LIN {X 0,Y 560.232,Z 513.242,A -85,B 0,C 180,E1 26436.285,E2 26436.285} C_VEL
LIN {X 0,Y 559.276,Z 513.366,A -85,B 0,C 180,E1 26435.497,E2 26435.497} C_VEL
LIN {X 0,Y 552.777,Z 514.194,A -85,B 0,C 180,E1 26433.228,E2 26433.228} C_VEL
LIN {X 0,Y 552.308,Z 514.247,A -85,B 0,C 180,E1 26432.709,E2 26432.709} C_VEL
LIN {X 0,Y 552.316,Z 514.235,A -85,B 0,C 180,E1 26429.509,E2 26429.509} C_VEL
LIN {X 0,Y 552.286,Z 514.241,A -85,B 0,C 180,E1 26426.2,E2 26426.2} C_VEL
LIN {X 0,Y 552.335,Z 514.246,A -85,B 0,C 180,E1 26422.97,E2 26422.97} C_VEL
LIN {X 0,Y 552.273,Z 514.249,A -85,B 0,C 180,E1 26419.735,E2 26419.735} C_VEL
LIN {X 0,Y 552.341,Z 514.249,A -85,B 0,C 180,E1 26416.537,E2 26416.537} C_VEL
LIN {X 0,Y 552.26,Z 514.237,A -85,B 0,C 180,E1 26413.329,E2 26413.329} C_VEL
LIN {X 0,Y 552.307,Z 514.386,A -85,B 0,C 180,E1 26411.845,E2 26411.845} C_VEL
LIN {X 0,Y 553.529,Z 517.662,A -85,B 0,C 180,E1 26411.676,E2 26411.676} C_VEL
LIN {X 0,Y 555.648,Z 520.327,A -85,B 0,C 180,E1 26411.436,E2 26411.436} C_VEL
LIN {X 0,Y 558.42,Z 524.351,A -85,B 0,C 180,E1 26411.118,E2 26411.118} C_VEL
LIN {X 0,Y 563.975,Z 533.241,A -85,B 0,C 180,E1 26410.48,E2 26410.48} C_VEL
LIN {X 0,Y 562.51,Z 710.248,A -85,B 0,C 180,E1 26407.75,E2 26407.75} C_VEL
LIN {X 0,Y 561.245,Z 862.07,A -85,B 0,C 180,E1 26405.443,E2 26405.443} C_VEL
LIN {X 0,Y 560.691,Z 885.823,A -85,B 0,C 180,E1 26404.892,E2 26404.892} C_VEL
LIN {X 0,Y 560.12,Z 907.981,A -85,B 0,C 180,E1 26404.188,E2 26404.188} C_VEL
LIN {X 0,Y 559.329,Z 930.017,A -85,B 0,C 180,E1 26403.285,E2 26403.285} C_VEL
LIN {X 0,Y 558.535,Z 951.055,A -85,B 0,C 180,E1 26402.24,E2 26402.24} C_VEL
LIN {X 0,Y 557.663,Z 971.471,A -85,B 0,C 180,E1 26401.015,E2 26401.015} C_VEL
LIN {X 0,Y 556.752,Z 991.835,A -85,B 0,C 180,E1 26399.595,E2 26399.595} C_VEL
LIN {X 0,Y 555.897,Z 1010.735,A -85,B 0,C 180,E1 26398.057,E2 26398.057} C_VEL
LIN {X 0,Y 555.048,Z 1029.466,A -85,B 0,C 180,E1 26396.305,E2 26396.305} C_VEL
LIN {X 0,Y 554.331,Z 1046.61,A -85,B 0,C 180,E1 26394.472,E2 26394.472} C_VEL
LIN {X 0,Y 553.671,Z 1062.502,A -85,B 0,C 180,E1 26392.51,E2 26392.51} C_VEL
LIN {X 0,Y 553.105,Z 1078.047,A -85,B 0,C 180,E1 26390.309,E2 26390.309} C_VEL
LIN {X 0,Y 552.695,Z 1090.742,A -85,B 0,C 180,E1 26388.239,E2 26388.239} C_VEL
LIN {X 0,Y 552.374,Z 1102.624,A -85,B 0,C 180,E1 26385.971,E2 26385.971} C_VEL
LIN {X 0,Y 552.165,Z 1112.707,A -85,B 0,C 180,E1 26383.723,E2 26383.723} C_VEL
LIN {X 0,Y 552.033,Z 1121.257,A -85,B 0,C 180,E1 26381.387,E2 26381.387} C_VEL
LIN {X 0,Y 551.968,Z 1128.186,A -85,B 0,C 180,E1 26379.068,E2 26379.068} C_VEL
LIN {X 0,Y 551.902,Z 1133.165,A -85,B 0,C 180,E1 26376.868,E2 26376.868} C_VEL
LIN {X 0,Y 551.907,Z 1136.995,A -85,B 0,C 180,E1 26374.572,E2 26374.572} C_VEL
LIN {X 0,Y 551.916,Z 1139.227,A -85,B 0,C 180,E1 26372.181,E2 26372.181} C_VEL
LIN {X 0,Y 551.901,Z 1139.971,A -85,B 0,C 180,E1 26369.793,E2 26369.793} C_VEL
LIN {X 0,Y 551.915,Z 1139.152,A -85,B 0,C 180,E1 26367.612,E2 26367.612} C_VEL
LIN {X 0,Y 551.904,Z 1136.823,A -85,B 0,C 180,E1 26365.22,E2 26365.22} C_VEL
LIN {X 0,Y 551.901,Z 1133.137,A -85,B 0,C 180,E1 26363.028,E2 26363.028} C_VEL
LIN {X 0,Y 551.967,Z 1128.151,A -85,B 0,C 180,E1 26360.828,E2 26360.828} C_VEL
LIN {X 0,Y 552.034,Z 1121.13,A -85,B 0,C 180,E1 26358.485,E2 26358.485} C_VEL
LIN {X 0,Y 552.166,Z 1112.641,A -85,B 0,C 180,E1 26356.171,E2 26356.171} C_VEL
LIN {X 0,Y 552.377,Z 1102.538,A -85,B 0,C 180,E1 26353.922,E2 26353.922} C_VEL
LIN {X 0,Y 552.697,Z 1090.632,A -85,B 0,C 180,E1 26351.653,E2 26351.653} C_VEL
LIN {X 0,Y 553.11,Z 1077.918,A -85,B 0,C 180,E1 26349.581,E2 26349.581} C_VEL
LIN {X 0,Y 553.675,Z 1062.338,A -85,B 0,C 180,E1 26347.378,E2 26347.378} C_VEL
LIN {X 0,Y 554.351,Z 1046.033,A -85,B 0,C 180,E1 26345.374,E2 26345.374} C_VEL
LIN {X 0,Y 555.077,Z 1028.825,A -85,B 0,C 180,E1 26343.54,E2 26343.54} C_VEL
LIN {X 0,Y 555.939,Z 1009.778,A -85,B 0,C 180,E1 26341.77,E2 26341.77} C_VEL
LIN {X 0,Y 556.804,Z 990.757,A -85,B 0,C 180,E1 26340.23,E2 26340.23} C_VEL
LIN {X 0,Y 557.691,Z 970.828,A -85,B 0,C 180,E1 26338.853,E2 26338.853} C_VEL
LIN {X 0,Y 558.581,Z 949.389,A -85,B 0,C 180,E1 26337.581,E2 26337.581} C_VEL
LIN {X 0,Y 559.362,Z 929.258,A -85,B 0,C 180,E1 26336.591,E2 26336.591} C_VEL
LIN {X 0,Y 560.139,Z 906.727,A -85,B 0,C 180,E1 26335.678,E2 26335.678} C_VEL
LIN {X 0,Y 560.713,Z 885.175,A -85,B 0,C 180,E1 26335,E2 26335} C_VEL
LIN {X 0,Y 561.252,Z 861.559,A -85,B 0,C 180,E1 26334.459,E2 26334.459} C_VEL
LIN {X 0,Y 562.929,Z 657.408,A -85,B 0,C 180,E1 26331.353,E2 26331.353} C_VEL
LIN {X 0,Y 563.852,Z 532.773,A -85,B 0,C 180,E1 26329.412,E2 26329.412} C_VEL
LIN {X 0,Y 557.609,Z 523.466,A -85,B 0,C 180,E1 26328.705,E2 26328.705} C_VEL
LIN {X 0,Y 554.774,Z 519.146,A -85,B 0,C 180,E1 26328.374,E2 26328.374} C_VEL
LIN {X 0,Y 552.748,Z 516.13,A -85,B 0,C 180,E1 26328.136,E2 26328.136} C_VEL
LIN {X 0,Y 552.289,Z 514.252,A -85,B 0,C 180,E1 26328.049,E2 26328.049} C_VEL
LIN {X 0,Y 552.263,Z 514.254,A -85,B 0,C 180,E1 26324.771,E2 26324.771} C_VEL
LIN {X 0,Y 552.297,Z 514.25,A -85,B 0,C 180,E1 26321.766,E2 26321.766} C_VEL
LIN {X 0,Y 552.274,Z 514.244,A -85,B 0,C 180,E1 26318.52,E2 26318.52} C_VEL
LIN {X 0,Y 552.315,Z 514.242,A -85,B 0,C 180,E1 26315.401,E2 26315.401} C_VEL
LIN {X 0,Y 552.279,Z 514.249,A -85,B 0,C 180,E1 26312.083,E2 26312.083} C_VEL
LIN {X 0,Y 552.34,Z 514.234,A -85,B 0,C 180,E1 26308.903,E2 26308.903} C_VEL
LIN {X 0,Y 552.288,Z 514.247,A -85,B 0,C 180,E1 26305.634,E2 26305.634} C_VEL
LIN {X 0,Y 552.345,Z 514.241,A -85,B 0,C 180,E1 26302.329,E2 26302.329} C_VEL
LIN {X 0,Y 552.304,Z 514.248,A -85,B 0,C 180,E1 26299.018,E2 26299.018} C_VEL
LIN {X 0,Y 552.313,Z 514.239,A -85,B 0,C 180,E1 26295.541,E2 26295.541} C_VEL
LIN {X 0,Y 552.342,Z 514.244,A -85,B 0,C 180,E1 26292.228,E2 26292.228} C_VEL
LIN {X 0,Y 552.307,Z 514.245,A -85,B 0,C 180,E1 26288.852,E2 26288.852} C_VEL
LIN {X 0,Y 552.335,Z 514.241,A -85,B 0,C 180,E1 26285.61,E2 26285.61} C_VEL
LIN {X 0,Y 552.32,Z 514.248,A -85,B 0,C 180,E1 26282.283,E2 26282.283} C_VEL
LIN {X 0,Y 552.338,Z 514.24,A -85,B 0,C 180,E1 26278.859,E2 26278.859} C_VEL
LIN {X 0,Y 552.333,Z 514.246,A -85,B 0,C 180,E1 26275.432,E2 26275.432} C_VEL
LIN {X 0,Y 552.325,Z 514.244,A -85,B 0,C 180,E1 26272.092,E2 26272.092} C_VEL
LIN {X 0,Y 552.321,Z 514.23,A -85,B 0,C 180,E1 26268.831,E2 26268.831} C_VEL
LIN {X 0,Y 552.34,Z 514.248,A -85,B 0,C 180,E1 26265.427,E2 26265.427} C_VEL
LIN {X 0,Y 552.338,Z 514.226,A -85,B 0,C 180,E1 26261.968,E2 26261.968} C_VEL
LIN {X 0,Y 552.317,Z 514.246,A -85,B 0,C 180,E1 26258.662,E2 26258.662} C_VEL
LIN {X 0,Y 552.336,Z 514.233,A -85,B 0,C 180,E1 26255.332,E2 26255.332} C_VEL
LIN {X 0,Y 552.303,Z 514.24,A -85,B 0,C 180,E1 26252.039,E2 26252.039} C_VEL
LIN {X 0,Y 552.341,Z 514.247,A -85,B 0,C 180,E1 26248.696,E2 26248.696} C_VEL
LIN {X 0,Y 552.315,Z 514.236,A -85,B 0,C 180,E1 26245.359,E2 26245.359} C_VEL
LIN {X 0,Y 552.3,Z 514.238,A -85,B 0,C 180,E1 26241.953,E2 26241.953} C_VEL
LIN {X 0,Y 552.343,Z 514.241,A -85,B 0,C 180,E1 26238.698,E2 26238.698} C_VEL
LIN {X 0,Y 552.285,Z 514.248,A -85,B 0,C 180,E1 26235.378,E2 26235.378} C_VEL
LIN {X 0,Y 552.359,Z 514.374,A -85,B 0,C 180,E1 26234.162,E2 26234.162} C_VEL
LIN {X 0,Y 553.707,Z 517.879,A -85,B 0,C 180,E1 26233.756,E2 26233.756} C_VEL
LIN {X 0,Y 560.161,Z 531.726,A -85,B 0,C 180,E1 26232.053,E2 26232.053} C_VEL
LIN {X 0,Y 561.65,Z 535.297,A -85,B 0,C 180,E1 26231.643,E2 26231.643} C_VEL
LIN {X 0,Y 561.544,Z 543.497,A -85,B 0,C 180,E1 26231.065,E2 26231.065} C_VEL
LIN {X 0,Y 564.073,Z 556.183,A -85,B 0,C 180,E1 26230.632,E2 26230.632} C_VEL
LIN {X 0,Y 562.534,Z 736.937,A -85,B 0,C 180,E1 26227.845,E2 26227.845} C_VEL
LIN {X 0,Y 561.249,Z 891.903,A -85,B 0,C 180,E1 26225.49,E2 26225.49} C_VEL
LIN {X 0,Y 560.693,Z 915.755,A -85,B 0,C 180,E1 26224.939,E2 26224.939} C_VEL
LIN {X 0,Y 560.119,Z 937.904,A -85,B 0,C 180,E1 26224.236,E2 26224.236} C_VEL
LIN {X 0,Y 559.343,Z 959.686,A -85,B 0,C 180,E1 26223.345,E2 26223.345} C_VEL
LIN {X 0,Y 558.544,Z 980.789,A -85,B 0,C 180,E1 26222.3,E2 26222.3} C_VEL
LIN {X 0,Y 557.68,Z 1001.05,A -85,B 0,C 180,E1 26221.088,E2 26221.088} C_VEL
LIN {X 0,Y 556.795,Z 1020.934,A -85,B 0,C 180,E1 26219.711,E2 26219.711} C_VEL
LIN {X 0,Y 555.952,Z 1039.506,A -85,B 0,C 180,E1 26218.208,E2 26218.208} C_VEL
LIN {X 0,Y 555.077,Z 1058.795,A -85,B 0,C 180,E1 26216.418,E2 26216.418} C_VEL
LIN {X 0,Y 554.365,Z 1075.664,A -85,B 0,C 180,E1 26214.622,E2 26214.622} C_VEL
LIN {X 0,Y 553.688,Z 1091.996,A -85,B 0,C 180,E1 26212.621,E2 26212.621} C_VEL
LIN {X 0,Y 553.14,Z 1106.921,A -85,B 0,C 180,E1 26210.529,E2 26210.529} C_VEL
LIN {X 0,Y 552.723,Z 1119.735,A -85,B 0,C 180,E1 26208.455,E2 26208.455} C_VEL
LIN {X 0,Y 552.396,Z 1131.8,A -85,B 0,C 180,E1 26206.185,E2 26206.185} C_VEL
LIN {X 0,Y 552.203,Z 1141.077,A -85,B 0,C 180,E1 26204.149,E2 26204.149} C_VEL
LIN {X 0,Y 552.052,Z 1150.342,A -85,B 0,C 180,E1 26201.704,E2 26201.704} C_VEL
LIN {X 0,Y 551.951,Z 1156.869,A -85,B 0,C 180,E1 26199.593,E2 26199.593} C_VEL
LIN {X 0,Y 551.902,Z 1162.635,A -85,B 0,C 180,E1 26197.181,E2 26197.181} C_VEL
LIN {X 0,Y 551.913,Z 1166.277,A -85,B 0,C 180,E1 26195.093,E2 26195.093} C_VEL
LIN {X 0,Y 551.91,Z 1168.988,A -85,B 0,C 180,E1 26192.596,E2 26192.596} C_VEL
LIN {X 0,Y 551.884,Z 1169.895,A -85,B 0,C 180,E1 26190.519,E2 26190.519} C_VEL
LIN {X 0,Y 551.908,Z 1169.391,A -85,B 0,C 180,E1 26188.027,E2 26188.027} C_VEL
LIN {X 0,Y 551.917,Z 1167.503,A -85,B 0,C 180,E1 26185.844,E2 26185.844} C_VEL
LIN {X 0,Y 551.917,Z 1163.667,A -85,B 0,C 180,E1 26183.342,E2 26183.342} C_VEL
LIN {X 0,Y 551.96,Z 1159.061,A -85,B 0,C 180,E1 26181.247,E2 26181.247} C_VEL
LIN {X 0,Y 552.018,Z 1152.118,A -85,B 0,C 180,E1 26178.825,E2 26178.825} C_VEL
LIN {X 0,Y 552.129,Z 1144.518,A -85,B 0,C 180,E1 26176.703,E2 26176.703} C_VEL
LIN {X 0,Y 552.341,Z 1134.399,A -85,B 0,C 180,E1 26174.352,E2 26174.352} C_VEL
LIN {X 0,Y 552.64,Z 1123.4,A -85,B 0,C 180,E1 26172.196,E2 26172.196} C_VEL
LIN {X 0,Y 553.038,Z 1110.462,A -85,B 0,C 180,E1 26170.019,E2 26170.019} C_VEL
LIN {X 0,Y 553.551,Z 1096.068,A -85,B 0,C 180,E1 26167.912,E2 26167.912} C_VEL
LIN {X 0,Y 554.162,Z 1080.256,A -85,B 0,C 180,E1 26165.917,E2 26165.917} C_VEL
LIN {X 0,Y 554.943,Z 1062.113,A -85,B 0,C 180,E1 26163.92,E2 26163.92} C_VEL
LIN {X 0,Y 555.763,Z 1043.892,A -85,B 0,C 180,E1 26162.169,E2 26162.169} C_VEL
LIN {X 0,Y 556.617,Z 1024.906,A -85,B 0,C 180,E1 26160.599,E2 26160.599} C_VEL
LIN {X 0,Y 557.562,Z 1003.711,A -85,B 0,C 180,E1 26159.084,E2 26159.084} C_VEL
LIN {X 0,Y 558.414,Z 983.89,A -85,B 0,C 180,E1 26157.878,E2 26157.878} C_VEL
LIN {X 0,Y 559.232,Z 962.227,A -85,B 0,C 180,E1 26156.77,E2 26156.77} C_VEL
LIN {X 0,Y 559.996,Z 941.495,A -85,B 0,C 180,E1 26155.9,E2 26155.9} C_VEL
LIN {X 0,Y 560.629,Z 918.213,A -85,B 0,C 180,E1 26155.13,E2 26155.13} C_VEL
LIN {X 0,Y 561.199,Z 895.627,A -85,B 0,C 180,E1 26154.578,E2 26154.578} C_VEL
LIN {X 0,Y 561.613,Z 853.941,A -85,B 0,C 180,E1 26153.917,E2 26153.917} C_VEL
LIN {X 0,Y 563.343,Z 644.147,A -85,B 0,C 180,E1 26150.737,E2 26150.737} C_VEL
LIN {X 0,Y 563.913,Z 554.474,A -85,B 0,C 180,E1 26149.326,E2 26149.326} C_VEL
LIN {X 0,Y 561.439,Z 542.402,A -85,B 0,C 180,E1 26148.878,E2 26148.878} C_VEL
LIN {X 0,Y 561.611,Z 534.829,A -85,B 0,C 180,E1 26148.318,E2 26148.318} C_VEL
LIN {X 0,Y 555.718,Z 522.083,A -85,B 0,C 180,E1 26146.776,E2 26146.776} C_VEL
LIN {X 0,Y 552.442,Z 514.864,A -85,B 0,C 180,E1 26145.885,E2 26145.885} C_VEL
LIN {X 0,Y 552.341,Z 514.227,A -85,B 0,C 180,E1 26145.794,E2 26145.794} C_VEL
LIN {X 0,Y 552.285,Z 514.244,A -85,B 0,C 180,E1 26142.537,E2 26142.537} C_VEL
LIN {X 0,Y 552.347,Z 514.246,A -85,B 0,C 180,E1 26139.314,E2 26139.314} C_VEL
LIN {X 0,Y 552.298,Z 514.25,A -85,B 0,C 180,E1 26136.041,E2 26136.041} C_VEL
LIN {X 0,Y 552.327,Z 514.243,A -85,B 0,C 180,E1 26132.646,E2 26132.646} C_VEL
LIN {X 0,Y 552.328,Z 514.235,A -85,B 0,C 180,E1 26129.378,E2 26129.378} C_VEL
LIN {X 0,Y 552.31,Z 514.243,A -85,B 0,C 180,E1 26125.982,E2 26125.982} C_VEL
LIN {X 0,Y 552.337,Z 514.239,A -85,B 0,C 180,E1 26122.679,E2 26122.679} C_VEL
LIN {X 0,Y 552.313,Z 514.244,A -85,B 0,C 180,E1 26119.407,E2 26119.407} C_VEL
LIN {X 0,Y 552.337,Z 514.238,A -85,B 0,C 180,E1 26116.079,E2 26116.079} C_VEL
LIN {X 0,Y 552.336,Z 514.242,A -85,B 0,C 180,E1 26112.649,E2 26112.649} C_VEL
LIN {X 0,Y 552.329,Z 514.235,A -85,B 0,C 180,E1 26109.271,E2 26109.271} C_VEL
LIN {X 0,Y 552.325,Z 514.243,A -85,B 0,C 180,E1 26105.922,E2 26105.922} C_VEL
LIN {X 0,Y 552.328,Z 514.246,A -85,B 0,C 180,E1 26102.594,E2 26102.594} C_VEL
LIN {X 0,Y 552.325,Z 514.241,A -85,B 0,C 180,E1 26099.274,E2 26099.274} C_VEL
LIN {X 0,Y 552.334,Z 514.247,A -85,B 0,C 180,E1 26095.847,E2 26095.847} C_VEL
LIN {X 0,Y 552.342,Z 514.241,A -85,B 0,C 180,E1 26092.511,E2 26092.511} C_VEL
LIN {X 0,Y 552.308,Z 514.234,A -85,B 0,C 180,E1 26089.148,E2 26089.148} C_VEL
LIN {X 0,Y 552.339,Z 514.245,A -85,B 0,C 180,E1 26085.855,E2 26085.855} C_VEL
LIN {X 0,Y 552.303,Z 514.228,A -85,B 0,C 180,E1 26082.566,E2 26082.566} C_VEL
LIN {X 0,Y 552.335,Z 514.249,A -85,B 0,C 180,E1 26079.218,E2 26079.218} C_VEL
LIN {X 0,Y 552.31,Z 514.228,A -85,B 0,C 180,E1 26075.963,E2 26075.963} C_VEL
LIN {X 0,Y 552.308,Z 514.247,A -85,B 0,C 180,E1 26072.709,E2 26072.709} C_VEL
LIN {X 0,Y 551.289,Z 514.37,A -85,B 0,C 180,E1 26071.91,E2 26071.91} C_VEL
LIN {X 0,Y 544.934,Z 515.153,A -85,B 0,C 180,E1 26069.666,E2 26069.666} C_VEL
LIN {X 0,Y 544.406,Z 515.225,A -85,B 0,C 180,E1 26069.082,E2 26069.082} C_VEL
LIN {X 0,Y 544.341,Z 515.228,A -85,B 0,C 180,E1 26065.928,E2 26065.928} C_VEL
LIN {X 0,Y 544.402,Z 515.237,A -85,B 0,C 180,E1 26062.68,E2 26062.68} C_VEL
LIN {X 0,Y 544.334,Z 515.238,A -85,B 0,C 180,E1 26059.505,E2 26059.505} C_VEL
LIN {X 0,Y 544.373,Z 515.242,A -85,B 0,C 180,E1 26056.176,E2 26056.176} C_VEL
LIN {X 0,Y 544.326,Z 515.223,A -85,B 0,C 180,E1 26053.104,E2 26053.104} C_VEL
LIN {X 0,Y 544.388,Z 515.369,A -85,B 0,C 180,E1 26052.58,E2 26052.58} C_VEL
LIN {X 0,Y 545.656,Z 518.647,A -85,B 0,C 180,E1 26052.4,E2 26052.4} C_VEL
LIN {X 0,Y 547.75,Z 521.261,A -85,B 0,C 180,E1 26052.154,E2 26052.154} C_VEL
LIN {X 0,Y 550.481,Z 525.313,A -85,B 0,C 180,E1 26051.828,E2 26051.828} C_VEL
LIN {X 0,Y 557.856,Z 536.647,A -85,B 0,C 180,E1 26050.962,E2 26050.962} C_VEL
LIN {X 0,Y 556.138,Z 716.399,A -85,B 0,C 180,E1 26048.162,E2 26048.162} C_VEL
LIN {X 0,Y 554.723,Z 862.114,A -85,B 0,C 180,E1 26045.923,E2 26045.923} C_VEL
LIN {X 0,Y 554.113,Z 885.625,A -85,B 0,C 180,E1 26045.375,E2 26045.375} C_VEL
LIN {X 0,Y 553.439,Z 907.468,A -85,B 0,C 180,E1 26044.679,E2 26044.679} C_VEL
LIN {X 0,Y 552.6,Z 928.745,A -85,B 0,C 180,E1 26043.807,E2 26043.807} C_VEL
LIN {X 0,Y 551.702,Z 948.86,A -85,B 0,C 180,E1 26042.812,E2 26042.812} C_VEL
LIN {X 0,Y 550.716,Z 969.39,A -85,B 0,C 180,E1 26041.593,E2 26041.593} C_VEL
LIN {X 0,Y 549.729,Z 988.993,A -85,B 0,C 180,E1 26040.238,E2 26040.238} C_VEL
LIN {X 0,Y 548.677,Z 1008.761,A -85,B 0,C 180,E1 26038.638,E2 26038.638} C_VEL
LIN {X 0,Y 547.668,Z 1027.888,A -85,B 0,C 180,E1 26036.855,E2 26036.855} C_VEL
LIN {X 0,Y 546.862,Z 1044.251,A -85,B 0,C 180,E1 26035.099,E2 26035.099} C_VEL
LIN {X 0,Y 546.058,Z 1060.805,A -85,B 0,C 180,E1 26033.07,E2 26033.07} C_VEL
LIN {X 0,Y 545.448,Z 1075.209,A -85,B 0,C 180,E1 26031.057,E2 26031.057} C_VEL
LIN {X 0,Y 544.92,Z 1088.839,A -85,B 0,C 180,E1 26028.841,E2 26028.841} C_VEL
LIN {X 0,Y 544.523,Z 1101.066,A -85,B 0,C 180,E1 26026.536,E2 26026.536} C_VEL
LIN {X 0,Y 544.266,Z 1110.885,A -85,B 0,C 180,E1 26024.36,E2 26024.36} C_VEL
LIN {X 0,Y 544.073,Z 1119.835,A -85,B 0,C 180,E1 26021.986,E2 26021.986} C_VEL
LIN {X 0,Y 543.966,Z 1126.376,A -85,B 0,C 180,E1 26019.864,E2 26019.864} C_VEL
LIN {X 0,Y 543.916,Z 1132.34,A -85,B 0,C 180,E1 26017.393,E2 26017.393} C_VEL
LIN {X 0,Y 543.909,Z 1136.049,A -85,B 0,C 180,E1 26015.274,E2 26015.274} C_VEL
LIN {X 0,Y 543.891,Z 1138.823,A -85,B 0,C 180,E1 26012.845,E2 26012.845} C_VEL
LIN {X 0,Y 543.885,Z 1139.863,A -85,B 0,C 180,E1 26010.632,E2 26010.632} C_VEL
LIN {X 0,Y 543.905,Z 1139.622,A -85,B 0,C 180,E1 26008.315,E2 26008.315} C_VEL
LIN {X 0,Y 543.914,Z 1137.778,A -85,B 0,C 180,E1 26005.995,E2 26005.995} C_VEL
LIN {X 0,Y 543.93,Z 1134.375,A -85,B 0,C 180,E1 26003.562,E2 26003.562} C_VEL
LIN {X 0,Y 543.962,Z 1129.68,A -85,B 0,C 180,E1 26001.331,E2 26001.331} C_VEL
LIN {X 0,Y 544.03,Z 1123.191,A -85,B 0,C 180,E1 25998.939,E2 25998.939} C_VEL
LIN {X 0,Y 544.162,Z 1115.1,A -85,B 0,C 180,E1 25996.614,E2 25996.614} C_VEL
LIN {X 0,Y 544.405,Z 1105.125,A -85,B 0,C 180,E1 25994.228,E2 25994.228} C_VEL
LIN {X 0,Y 544.742,Z 1094.22,A -85,B 0,C 180,E1 25992.04,E2 25992.04} C_VEL
LIN {X 0,Y 545.227,Z 1080.747,A -85,B 0,C 180,E1 25989.721,E2 25989.721} C_VEL
LIN {X 0,Y 545.824,Z 1066.534,A -85,B 0,C 180,E1 25987.603,E2 25987.603} C_VEL
LIN {X 0,Y 546.546,Z 1050.45,A -85,B 0,C 180,E1 25985.539,E2 25985.539} C_VEL
LIN {X 0,Y 547.459,Z 1032.181,A -85,B 0,C 180,E1 25983.498,E2 25983.498} C_VEL
LIN {X 0,Y 548.433,Z 1013.806,A -85,B 0,C 180,E1 25981.711,E2 25981.711} C_VEL
LIN {X 0,Y 549.387,Z 995.155,A -85,B 0,C 180,E1 25980.148,E2 25980.148} C_VEL
LIN {X 0,Y 550.495,Z 973.923,A -85,B 0,C 180,E1 25978.612,E2 25978.612} C_VEL
LIN {X 0,Y 551.439,Z 954.553,A -85,B 0,C 180,E1 25977.417,E2 25977.417} C_VEL
LIN {X 0,Y 552.455,Z 931.886,A -85,B 0,C 180,E1 25976.246,E2 25976.246} C_VEL
LIN {X 0,Y 553.28,Z 911.823,A -85,B 0,C 180,E1 25975.396,E2 25975.396} C_VEL
LIN {X 0,Y 554.017,Z 888.332,A -85,B 0,C 180,E1 25974.611,E2 25974.611} C_VEL
LIN {X 0,Y 554.667,Z 865.768,A -85,B 0,C 180,E1 25974.055,E2 25974.055} C_VEL
LIN {X 0,Y 555.136,Z 825.273,A -85,B 0,C 180,E1 25973.404,E2 25973.404} C_VEL
LIN {X 0,Y 557.18,Z 611.78,A -85,B 0,C 180,E1 25970.134,E2 25970.134} C_VEL
LIN {X 0,Y 557.707,Z 536.226,A -85,B 0,C 180,E1 25968.927,E2 25968.927} C_VEL
LIN {X 0,Y 549.513,Z 524.202,A -85,B 0,C 180,E1 25967.973,E2 25967.973} C_VEL
LIN {X 0,Y 546.885,Z 520.112,A -85,B 0,C 180,E1 25967.653,E2 25967.653} C_VEL
LIN {X 0,Y 544.828,Z 517.102,A -85,B 0,C 180,E1 25967.404,E2 25967.404} C_VEL
LIN {X 0,Y 544.355,Z 515.24,A -85,B 0,C 180,E1 25967.318,E2 25967.318} C_VEL
LIN {X 0,Y 544.327,Z 515.244,A -85,B 0,C 180,E1 25964.244,E2 25964.244} C_VEL
LIN {X 0,Y 544.345,Z 515.239,A -85,B 0,C 180,E1 25960.82,E2 25960.82} C_VEL
LIN {X 0,Y 544.342,Z 515.234,A -85,B 0,C 180,E1 25957.83,E2 25957.83} C_VEL
LIN {X 0,Y 544.342,Z 515.225,A -85,B 0,C 180,E1 25954.326,E2 25954.326} C_VEL
LIN {X 0,Y 544.383,Z 515.237,A -85,B 0,C 180,E1 25951.195,E2 25951.195} C_VEL
LIN {X 0,Y 544.346,Z 515.232,A -85,B 0,C 180,E1 25947.93,E2 25947.93} C_VEL
LIN {X 0,Y 544.399,Z 515.224,A -85,B 0,C 180,E1 25944.756,E2 25944.756} C_VEL
LIN {X 0,Y 544.354,Z 515.233,A -85,B 0,C 180,E1 25941.44,E2 25941.44} C_VEL
LIN {X 0,Y 544.401,Z 515.218,A -85,B 0,C 180,E1 25938.083,E2 25938.083} C_VEL
LIN {X 0,Y 544.372,Z 515.232,A -85,B 0,C 180,E1 25934.792,E2 25934.792} C_VEL
LIN {X 0,Y 544.379,Z 515.23,A -85,B 0,C 180,E1 25931.334,E2 25931.334} C_VEL
LIN {X 0,Y 544.404,Z 515.234,A -85,B 0,C 180,E1 25928.024,E2 25928.024} C_VEL
LIN {X 0,Y 544.373,Z 515.231,A -85,B 0,C 180,E1 25924.636,E2 25924.636} C_VEL
LIN {X 0,Y 544.399,Z 515.227,A -85,B 0,C 180,E1 25921.263,E2 25921.263} C_VEL
LIN {X 0,Y 544.399,Z 515.234,A -85,B 0,C 180,E1 25917.79,E2 25917.79} C_VEL
LIN {X 0,Y 544.389,Z 515.23,A -85,B 0,C 180,E1 25914.414,E2 25914.414} C_VEL
LIN {X 0,Y 544.387,Z 515.23,A -85,B 0,C 180,E1 25911.125,E2 25911.125} C_VEL
LIN {X 0,Y 544.39,Z 515.219,A -85,B 0,C 180,E1 25907.716,E2 25907.716} C_VEL
LIN {X 0,Y 544.39,Z 515.229,A -85,B 0,C 180,E1 25904.337,E2 25904.337} C_VEL
LIN {X 0,Y 544.389,Z 515.23,A -85,B 0,C 180,E1 25900.918,E2 25900.918} C_VEL
LIN {X 0,Y 544.399,Z 515.231,A -85,B 0,C 180,E1 25897.542,E2 25897.542} C_VEL
LIN {X 0,Y 544.37,Z 515.235,A -85,B 0,C 180,E1 25894.158,E2 25894.158} C_VEL
LIN {X 0,Y 544.402,Z 515.222,A -85,B 0,C 180,E1 25890.738,E2 25890.738} C_VEL
LIN {X 0,Y 544.391,Z 515.232,A -85,B 0,C 180,E1 25887.318,E2 25887.318} C_VEL
LIN {X 0,Y 544.36,Z 515.238,A -85,B 0,C 180,E1 25883.918,E2 25883.918} C_VEL
LIN {X 0,Y 544.406,Z 515.226,A -85,B 0,C 180,E1 25880.643,E2 25880.643} C_VEL
LIN {X 0,Y 544.348,Z 515.231,A -85,B 0,C 180,E1 25877.439,E2 25877.439} C_VEL
LIN {X 0,Y 544.382,Z 515.383,A -85,B 0,C 180,E1 25874.868,E2 25874.868} C_VEL
LIN {X 0,Y 545.474,Z 518.362,A -85,B 0,C 180,E1 25874.518,E2 25874.518} C_VEL
LIN {X 0,Y 552.146,Z 532.183,A -85,B 0,C 180,E1 25872.771,E2 25872.771} C_VEL
LIN {X 0,Y 555.117,Z 538.763,A -85,B 0,C 180,E1 25871.976,E2 25871.976} C_VEL
LIN {X 0,Y 555.123,Z 543.668,A -85,B 0,C 180,E1 25871.642,E2 25871.642} C_VEL
LIN {X 0,Y 557.98,Z 557.994,A -85,B 0,C 180,E1 25871.141,E2 25871.141} C_VEL
LIN {X 0,Y 556.197,Z 739.052,A -85,B 0,C 180,E1 25868.32,E2 25868.32} C_VEL
LIN {X 0,Y 554.726,Z 892.068,A -85,B 0,C 180,E1 25865.969,E2 25865.969} C_VEL
LIN {X 0,Y 554.111,Z 915.623,A -85,B 0,C 180,E1 25865.42,E2 25865.42} C_VEL
LIN {X 0,Y 553.438,Z 937.423,A -85,B 0,C 180,E1 25864.726,E2 25864.726} C_VEL
LIN {X 0,Y 552.598,Z 958.774,A -85,B 0,C 180,E1 25863.85,E2 25863.85} C_VEL
LIN {X 0,Y 551.714,Z 978.564,A -85,B 0,C 180,E1 25862.873,E2 25862.873} C_VEL
LIN {X 0,Y 550.684,Z 1000.062,A -85,B 0,C 180,E1 25861.595,E2 25861.595} C_VEL
LIN {X 0,Y 549.669,Z 1020.19,A -85,B 0,C 180,E1 25860.196,E2 25860.196} C_VEL
LIN {X 0,Y 548.621,Z 1039.87,A -85,B 0,C 180,E1 25858.587,E2 25858.587} C_VEL
LIN {X 0,Y 547.595,Z 1059.198,A -85,B 0,C 180,E1 25856.765,E2 25856.765} C_VEL
LIN {X 0,Y 546.766,Z 1076.398,A -85,B 0,C 180,E1 25854.904,E2 25854.904} C_VEL
LIN {X 0,Y 545.99,Z 1092.365,A -85,B 0,C 180,E1 25852.909,E2 25852.909} C_VEL
LIN {X 0,Y 545.329,Z 1107.631,A -85,B 0,C 180,E1 25850.724,E2 25850.724} C_VEL
LIN {X 0,Y 544.857,Z 1120.369,A -85,B 0,C 180,E1 25848.621,E2 25848.621} C_VEL
LIN {X 0,Y 544.476,Z 1132.322,A -85,B 0,C 180,E1 25846.318,E2 25846.318} C_VEL
LIN {X 0,Y 544.23,Z 1142.337,A -85,B 0,C 180,E1 25844.062,E2 25844.062} C_VEL
LIN {X 0,Y 544.072,Z 1150.699,A -85,B 0,C 180,E1 25841.77,E2 25841.77} C_VEL
LIN {X 0,Y 543.962,Z 1157.475,A -85,B 0,C 180,E1 25839.522,E2 25839.522} C_VEL
LIN {X 0,Y 543.904,Z 1162.841,A -85,B 0,C 180,E1 25837.181,E2 25837.181} C_VEL
LIN {X 0,Y 543.913,Z 1166.436,A -85,B 0,C 180,E1 25835.062,E2 25835.062} C_VEL
LIN {X 0,Y 543.913,Z 1169.056,A -85,B 0,C 180,E1 25832.528,E2 25832.528} C_VEL
LIN {X 0,Y 543.892,Z 1169.939,A -85,B 0,C 180,E1 25830.316,E2 25830.316} C_VEL
LIN {X 0,Y 543.913,Z 1169.324,A -85,B 0,C 180,E1 25827.893,E2 25827.893} C_VEL
LIN {X 0,Y 543.913,Z 1167.389,A -85,B 0,C 180,E1 25825.677,E2 25825.677} C_VEL
LIN {X 0,Y 543.913,Z 1163.667,A -85,B 0,C 180,E1 25823.243,E2 25823.243} C_VEL
LIN {X 0,Y 543.968,Z 1159.061,A -85,B 0,C 180,E1 25821.118,E2 25821.118} C_VEL
LIN {X 0,Y 544.042,Z 1152.117,A -85,B 0,C 180,E1 25818.659,E2 25818.659} C_VEL
LIN {X 0,Y 544.169,Z 1144.519,A -85,B 0,C 180,E1 25816.505,E2 25816.505} C_VEL
LIN {X 0,Y 544.418,Z 1134.398,A -85,B 0,C 180,E1 25814.118,E2 25814.118} C_VEL
LIN {X 0,Y 544.747,Z 1123.982,A -85,B 0,C 180,E1 25812.039,E2 25812.039} C_VEL
LIN {X 0,Y 545.237,Z 1110.463,A -85,B 0,C 180,E1 25809.721,E2 25809.721} C_VEL
LIN {X 0,Y 545.839,Z 1096.214,A -85,B 0,C 180,E1 25807.603,E2 25807.603} C_VEL
LIN {X 0,Y 546.549,Z 1080.405,A -85,B 0,C 180,E1 25805.578,E2 25805.578} C_VEL
LIN {X 0,Y 547.461,Z 1062.113,A -85,B 0,C 180,E1 25803.536,E2 25803.536} C_VEL
LIN {X 0,Y 548.428,Z 1043.894,A -85,B 0,C 180,E1 25801.764,E2 25801.764} C_VEL
LIN {X 0,Y 549.413,Z 1024.594,A -85,B 0,C 180,E1 25800.149,E2 25800.149} C_VEL
LIN {X 0,Y 550.535,Z 1003.114,A -85,B 0,C 180,E1 25798.604,E2 25798.604} C_VEL
LIN {X 0,Y 551.474,Z 983.813,A -85,B 0,C 180,E1 25797.419,E2 25797.419} C_VEL
LIN {X 0,Y 552.438,Z 962.229,A -85,B 0,C 180,E1 25796.307,E2 25796.307} C_VEL
LIN {X 0,Y 553.254,Z 942.438,A -85,B 0,C 180,E1 25795.466,E2 25795.466} C_VEL
LIN {X 0,Y 554.01,Z 918.686,A -85,B 0,C 180,E1 25794.666,E2 25794.666} C_VEL
LIN {X 0,Y 554.636,Z 896.601,A -85,B 0,C 180,E1 25794.118,E2 25794.118} C_VEL
LIN {X 0,Y 555.082,Z 861.165,A -85,B 0,C 180,E1 25793.538,E2 25793.538} C_VEL
LIN {X 0,Y 557.019,Z 655.677,A -85,B 0,C 180,E1 25790.393,E2 25790.393} C_VEL
LIN {X 0,Y 557.821,Z 556.252,A -85,B 0,C 180,E1 25788.815,E2 25788.815} C_VEL
LIN {X 0,Y 554.985,Z 542.47,A -85,B 0,C 180,E1 25788.299,E2 25788.299} C_VEL
LIN {X 0,Y 555.02,Z 538.523,A -85,B 0,C 180,E1 25787.996,E2 25787.996} C_VEL
LIN {X 0,Y 547.492,Z 522.549,A -85,B 0,C 180,E1 25786.016,E2 25786.016} C_VEL
LIN {X 0,Y 545.476,Z 518.351,A -85,B 0,C 180,E1 25785.482,E2 25785.482} C_VEL
LIN {X 0,Y 544.357,Z 515.223,A -85,B 0,C 180,E1 25785.079,E2 25785.079} C_VEL
LIN {X 0,Y 544.378,Z 515.226,A -85,B 0,C 180,E1 25781.938,E2 25781.938} C_VEL
LIN {X 0,Y 544.359,Z 515.238,A -85,B 0,C 180,E1 25778.645,E2 25778.645} C_VEL
LIN {X 0,Y 544.402,Z 515.228,A -85,B 0,C 180,E1 25775.347,E2 25775.347} C_VEL
LIN {X 0,Y 544.36,Z 515.235,A -85,B 0,C 180,E1 25772.061,E2 25772.061} C_VEL
LIN {X 0,Y 544.403,Z 515.222,A -85,B 0,C 180,E1 25768.763,E2 25768.763} C_VEL
LIN {X 0,Y 544.376,Z 515.236,A -85,B 0,C 180,E1 25765.454,E2 25765.454} C_VEL
LIN {X 0,Y 544.383,Z 515.227,A -85,B 0,C 180,E1 25761.946,E2 25761.946} C_VEL
LIN {X 0,Y 544.396,Z 515.219,A -85,B 0,C 180,E1 25758.61,E2 25758.61} C_VEL
LIN {X 0,Y 544.378,Z 515.231,A -85,B 0,C 180,E1 25755.227,E2 25755.227} C_VEL
LIN {X 0,Y 544.395,Z 515.219,A -85,B 0,C 180,E1 25751.87,E2 25751.87} C_VEL
LIN {X 0,Y 544.399,Z 515.232,A -85,B 0,C 180,E1 25748.449,E2 25748.449} C_VEL
LIN {X 0,Y 544.394,Z 515.227,A -85,B 0,C 180,E1 25745.057,E2 25745.057} C_VEL
LIN {X 0,Y 544.384,Z 515.233,A -85,B 0,C 180,E1 25741.684,E2 25741.684} C_VEL
LIN {X 0,Y 544.392,Z 515.233,A -85,B 0,C 180,E1 25738.421,E2 25738.421} C_VEL
LIN {X 0,Y 544.383,Z 515.228,A -85,B 0,C 180,E1 25735.048,E2 25735.048} C_VEL
LIN {X 0,Y 544.387,Z 515.23,A -85,B 0,C 180,E1 25731.551,E2 25731.551} C_VEL
LIN {X 0,Y 544.399,Z 515.219,A -85,B 0,C 180,E1 25728.129,E2 25728.129} C_VEL
LIN {X 0,Y 544.365,Z 515.232,A -85,B 0,C 180,E1 25724.881,E2 25724.881} C_VEL
LIN {X 0,Y 544.401,Z 515.217,A -85,B 0,C 180,E1 25721.585,E2 25721.585} C_VEL
LIN {X 0,Y 544.362,Z 515.233,A -85,B 0,C 180,E1 25718.334,E2 25718.334} C_VEL
LIN {X 0,Y 544.378,Z 515.23,A -85,B 0,C 180,E1 25714.891,E2 25714.891} C_VEL
LIN {X 0,Y 544.38,Z 515.231,A -85,B 0,C 180,E1 25711.616,E2 25711.616} C_VEL
LIN {X 0,Y 544.406,Z 515.225,A -85,B 0,C 180,E1 25709.082,E2 25709.082} C_VEL
LIN {X 0,Y 543.393,Z 515.361,A -85,B 0,C 180,E1 25708.271,E2 25708.271} C_VEL
LIN {X 0,Y 536.922,Z 516.154,A -85,B 0,C 180,E1 25705.995,E2 25705.995} C_VEL
LIN {X 0,Y 536.425,Z 516.212,A -85,B 0,C 180,E1 25705.402,E2 25705.402} C_VEL
LIN {X 0,Y 536.405,Z 516.223,A -85,B 0,C 180,E1 25702.039,E2 25702.039} C_VEL
LIN {X 0,Y 536.428,Z 516.226,A -85,B 0,C 180,E1 25698.997,E2 25698.997} C_VEL
LIN {X 0,Y 536.393,Z 516.232,A -85,B 0,C 180,E1 25695.652,E2 25695.652} C_VEL
LIN {X 0,Y 536.405,Z 516.378,A -85,B 0,C 180,E1 25693.358,E2 25693.358} C_VEL
LIN {X 0,Y 537.628,Z 519.602,A -85,B 0,C 180,E1 25693.176,E2 25693.176} C_VEL
LIN {X 0,Y 540.024,Z 522.465,A -85,B 0,C 180,E1 25692.884,E2 25692.884} C_VEL
LIN {X 0,Y 551.778,Z 540.074,A -85,B 0,C 180,E1 25691.455,E2 25691.455} C_VEL
LIN {X 0,Y 549.787,Z 723.474,A -85,B 0,C 180,E1 25688.569,E2 25688.569} C_VEL
LIN {X 0,Y 548.24,Z 862.265,A -85,B 0,C 180,E1 25686.414,E2 25686.414} C_VEL
LIN {X 0,Y 547.568,Z 885.607,A -85,B 0,C 180,E1 25685.864,E2 25685.864} C_VEL
LIN {X 0,Y 546.792,Z 907.386,A -85,B 0,C 180,E1 25685.167,E2 25685.167} C_VEL
LIN {X 0,Y 545.83,Z 929.195,A -85,B 0,C 180,E1 25684.262,E2 25684.262} C_VEL
LIN {X 0,Y 544.793,Z 949.997,A -85,B 0,C 180,E1 25683.219,E2 25683.219} C_VEL
LIN {X 0,Y 543.66,Z 970.388,A -85,B 0,C 180,E1 25681.984,E2 25681.984} C_VEL
LIN {X 0,Y 542.524,Z 990.378,A -85,B 0,C 180,E1 25680.575,E2 25680.575} C_VEL
LIN {X 0,Y 541.357,Z 1009.433,A -85,B 0,C 180,E1 25679.001,E2 25679.001} C_VEL
LIN {X 0,Y 540.205,Z 1028.687,A -85,B 0,C 180,E1 25677.171,E2 25677.171} C_VEL
LIN {X 0,Y 539.244,Z 1045.844,A -85,B 0,C 180,E1 25675.295,E2 25675.295} C_VEL
LIN {X 0,Y 538.356,Z 1061.664,A -85,B 0,C 180,E1 25673.303,E2 25673.303} C_VEL
LIN {X 0,Y 537.619,Z 1076.642,A -85,B 0,C 180,E1 25671.15,E2 25671.15} C_VEL
LIN {X 0,Y 537.063,Z 1089.477,A -85,B 0,C 180,E1 25669.014,E2 25669.014} C_VEL
LIN {X 0,Y 536.61,Z 1101.592,A -85,B 0,C 180,E1 25666.676,E2 25666.676} C_VEL
LIN {X 0,Y 536.315,Z 1111.346,A -85,B 0,C 180,E1 25664.467,E2 25664.467} C_VEL
LIN {X 0,Y 536.094,Z 1120.195,A -85,B 0,C 180,E1 25662.058,E2 25662.058} C_VEL
LIN {X 0,Y 535.976,Z 1126.741,A -85,B 0,C 180,E1 25659.883,E2 25659.883} C_VEL
LIN {X 0,Y 535.919,Z 1132.548,A -85,B 0,C 180,E1 25657.397,E2 25657.397} C_VEL
LIN {X 0,Y 535.911,Z 1136.209,A -85,B 0,C 180,E1 25655.246,E2 25655.246} C_VEL
LIN {X 0,Y 535.896,Z 1138.891,A -85,B 0,C 180,E1 25652.781,E2 25652.781} C_VEL
LIN {X 0,Y 535.885,Z 1139.863,A -85,B 0,C 180,E1 25650.642,E2 25650.642} C_VEL
LIN {X 0,Y 535.905,Z 1139.621,A -85,B 0,C 180,E1 25648.29,E2 25648.29} C_VEL
LIN {X 0,Y 535.916,Z 1137.777,A -85,B 0,C 180,E1 25645.935,E2 25645.935} C_VEL
LIN {X 0,Y 535.93,Z 1134.374,A -85,B 0,C 180,E1 25643.466,E2 25643.466} C_VEL
LIN {X 0,Y 535.969,Z 1129.679,A -85,B 0,C 180,E1 25641.201,E2 25641.201} C_VEL
LIN {X 0,Y 536.048,Z 1123.323,A -85,B 0,C 180,E1 25638.815,E2 25638.815} C_VEL
LIN {X 0,Y 536.196,Z 1115.507,A -85,B 0,C 180,E1 25636.521,E2 25636.521} C_VEL
LIN {X 0,Y 536.465,Z 1106.149,A -85,B 0,C 180,E1 25634.21,E2 25634.21} C_VEL
LIN {X 0,Y 536.835,Z 1095.379,A -85,B 0,C 180,E1 25631.991,E2 25631.991} C_VEL
LIN {X 0,Y 537.382,Z 1082.142,A -85,B 0,C 180,E1 25629.639,E2 25629.639} C_VEL
LIN {X 0,Y 537.997,Z 1068.866,A -85,B 0,C 180,E1 25627.605,E2 25627.605} C_VEL
LIN {X 0,Y 538.845,Z 1052.624,A -85,B 0,C 180,E1 25625.44,E2 25625.44} C_VEL
LIN {X 0,Y 539.819,Z 1035.856,A -85,B 0,C 180,E1 25623.488,E2 25623.488} C_VEL
LIN {X 0,Y 540.833,Z 1018.034,A -85,B 0,C 180,E1 25621.693,E2 25621.693} C_VEL
LIN {X 0,Y 542.049,Z 997.997,A -85,B 0,C 180,E1 25619.941,E2 25619.941} C_VEL
LIN {X 0,Y 543.222,Z 978.266,A -85,B 0,C 180,E1 25618.452,E2 25618.452} C_VEL
LIN {X 0,Y 544.379,Z 957.553,A -85,B 0,C 180,E1 25617.129,E2 25617.129} C_VEL
LIN {X 0,Y 545.488,Z 936.241,A -85,B 0,C 180,E1 25615.974,E2 25615.974} C_VEL
LIN {X 0,Y 546.446,Z 915.434,A -85,B 0,C 180,E1 25615.058,E2 25615.058} C_VEL
LIN {X 0,Y 547.344,Z 893.181,A -85,B 0,C 180,E1 25614.265,E2 25614.265} C_VEL
LIN {X 0,Y 547.976,Z 871.021,A -85,B 0,C 180,E1 25613.678,E2 25613.678} C_VEL
LIN {X 0,Y 548.523,Z 843.808,A -85,B 0,C 180,E1 25613.188,E2 25613.188} C_VEL
LIN {X 0,Y 550.69,Z 639.161,A -85,B 0,C 180,E1 25610.026,E2 25610.026} C_VEL
LIN {X 0,Y 551.608,Z 539.62,A -85,B 0,C 180,E1 25608.431,E2 25608.431} C_VEL
LIN {X 0,Y 541.844,Z 525.402,A -85,B 0,C 180,E1 25607.259,E2 25607.259} C_VEL
LIN {X 0,Y 539.257,Z 521.436,A -85,B 0,C 180,E1 25606.931,E2 25606.931} C_VEL
LIN {X 0,Y 537.046,Z 518.583,A -85,B 0,C 180,E1 25606.657,E2 25606.657} C_VEL
LIN {X 0,Y 536.378,Z 516.236,A -85,B 0,C 180,E1 25606.54,E2 25606.54} C_VEL
LIN {X 0,Y 536.436,Z 516.229,A -85,B 0,C 180,E1 25603.216,E2 25603.216} C_VEL
LIN {X 0,Y 536.39,Z 516.228,A -85,B 0,C 180,E1 25600.159,E2 25600.159} C_VEL
LIN {X 0,Y 536.44,Z 516.226,A -85,B 0,C 180,E1 25596.882,E2 25596.882} C_VEL
LIN {X 0,Y 536.405,Z 516.215,A -85,B 0,C 180,E1 25593.743,E2 25593.743} C_VEL
LIN {X 0,Y 536.424,Z 516.215,A -85,B 0,C 180,E1 25590.34,E2 25590.34} C_VEL
LIN {X 0,Y 536.432,Z 516.224,A -85,B 0,C 180,E1 25587.172,E2 25587.172} C_VEL
LIN {X 0,Y 536.414,Z 516.207,A -85,B 0,C 180,E1 25583.742,E2 25583.742} C_VEL
LIN {X 0,Y 536.467,Z 516.226,A -85,B 0,C 180,E1 25580.511,E2 25580.511} C_VEL
LIN {X 0,Y 536.419,Z 516.207,A -85,B 0,C 180,E1 25577.128,E2 25577.128} C_VEL
LIN {X 0,Y 536.465,Z 516.221,A -85,B 0,C 180,E1 25573.802,E2 25573.802} C_VEL
LIN {X 0,Y 536.45,Z 516.226,A -85,B 0,C 180,E1 25570.416,E2 25570.416} C_VEL
LIN {X 0,Y 536.437,Z 516.222,A -85,B 0,C 180,E1 25566.959,E2 25566.959} C_VEL
LIN {X 0,Y 536.458,Z 516.224,A -85,B 0,C 180,E1 25563.633,E2 25563.633} C_VEL
LIN {X 0,Y 536.441,Z 516.219,A -85,B 0,C 180,E1 25560.321,E2 25560.321} C_VEL
LIN {X 0,Y 536.46,Z 516.217,A -85,B 0,C 180,E1 25556.902,E2 25556.902} C_VEL
LIN {X 0,Y 536.457,Z 516.224,A -85,B 0,C 180,E1 25553.423,E2 25553.423} C_VEL
LIN {X 0,Y 536.45,Z 516.217,A -85,B 0,C 180,E1 25550.018,E2 25550.018} C_VEL
LIN {X 0,Y 536.446,Z 516.22,A -85,B 0,C 180,E1 25546.637,E2 25546.637} C_VEL
LIN {X 0,Y 536.459,Z 516.209,A -85,B 0,C 180,E1 25543.209,E2 25543.209} C_VEL
LIN {X 0,Y 536.461,Z 516.22,A -85,B 0,C 180,E1 25539.717,E2 25539.717} C_VEL
LIN {X 0,Y 536.43,Z 516.208,A -85,B 0,C 180,E1 25536.376,E2 25536.376} C_VEL
LIN {X 0,Y 536.463,Z 516.226,A -85,B 0,C 180,E1 25532.95,E2 25532.95} C_VEL
LIN {X 0,Y 536.435,Z 516.218,A -85,B 0,C 180,E1 25529.653,E2 25529.653} C_VEL
LIN {X 0,Y 536.426,Z 516.211,A -85,B 0,C 180,E1 25526.13,E2 25526.13} C_VEL
LIN {X 0,Y 536.464,Z 516.22,A -85,B 0,C 180,E1 25522.853,E2 25522.853} C_VEL
LIN {X 0,Y 536.413,Z 516.228,A -85,B 0,C 180,E1 25519.508,E2 25519.508} C_VEL
LIN {X 0,Y 536.457,Z 516.227,A -85,B 0,C 180,E1 25516.162,E2 25516.162} C_VEL
LIN {X 0,Y 536.449,Z 516.483,A -85,B 0,C 180,E1 25515.592,E2 25515.592} C_VEL
LIN {X 0,Y 537.713,Z 519.709,A -85,B 0,C 180,E1 25515.192,E2 25515.192} C_VEL
LIN {X 0,Y 545.846,Z 536.441,A -85,B 0,C 180,E1 25513.041,E2 25513.041} C_VEL
LIN {X 0,Y 548.615,Z 543.117,A -85,B 0,C 180,E1 25512.259,E2 25512.259} C_VEL
LIN {X 0,Y 551.933,Z 559.774,A -85,B 0,C 180,E1 25511.662,E2 25511.662} C_VEL
LIN {X 0,Y 549.897,Z 741.47,A -85,B 0,C 180,E1 25508.801,E2 25508.801} C_VEL
LIN {X 0,Y 548.243,Z 892.161,A -85,B 0,C 180,E1 25506.461,E2 25506.461} C_VEL
LIN {X 0,Y 547.571,Z 915.491,A -85,B 0,C 180,E1 25505.912,E2 25505.912} C_VEL
LIN {X 0,Y 546.795,Z 937.135,A -85,B 0,C 180,E1 25505.221,E2 25505.221} C_VEL
LIN {X 0,Y 545.868,Z 958.396,A -85,B 0,C 180,E1 25504.344,E2 25504.344} C_VEL
LIN {X 0,Y 544.92,Z 977.449,A -85,B 0,C 180,E1 25503.399,E2 25503.399} C_VEL
LIN {X 0,Y 543.719,Z 999.248,A -85,B 0,C 180,E1 25502.103,E2 25502.103} C_VEL
LIN {X 0,Y 542.585,Z 1019.406,A -85,B 0,C 180,E1 25500.694,E2 25500.694} C_VEL
LIN {X 0,Y 541.365,Z 1039.272,A -85,B 0,C 180,E1 25499.061,E2 25499.061} C_VEL
LIN {X 0,Y 540.199,Z 1058.792,A -85,B 0,C 180,E1 25497.205,E2 25497.205} C_VEL
LIN {X 0,Y 539.251,Z 1075.662,A -85,B 0,C 180,E1 25495.36,E2 25495.36} C_VEL
LIN {X 0,Y 538.339,Z 1091.996,A -85,B 0,C 180,E1 25493.304,E2 25493.304} C_VEL
LIN {X 0,Y 537.603,Z 1106.925,A -85,B 0,C 180,E1 25491.15,E2 25491.15} C_VEL
LIN {X 0,Y 537.052,Z 1119.732,A -85,B 0,C 180,E1 25489.014,E2 25489.014} C_VEL
LIN {X 0,Y 536.6,Z 1131.802,A -85,B 0,C 180,E1 25486.675,E2 25486.675} C_VEL
LIN {X 0,Y 536.312,Z 1141.534,A -85,B 0,C 180,E1 25484.467,E2 25484.467} C_VEL
LIN {X 0,Y 536.096,Z 1150.344,A -85,B 0,C 180,E1 25482.057,E2 25482.057} C_VEL
LIN {X 0,Y 535.975,Z 1156.868,A -85,B 0,C 180,E1 25479.882,E2 25479.882} C_VEL
LIN {X 0,Y 535.917,Z 1162.635,A -85,B 0,C 180,E1 25477.396,E2 25477.396} C_VEL
LIN {X 0,Y 535.913,Z 1166.277,A -85,B 0,C 180,E1 25475.245,E2 25475.245} C_VEL
LIN {X 0,Y 535.898,Z 1168.92,A -85,B 0,C 180,E1 25472.78,E2 25472.78} C_VEL
LIN {X 0,Y 535.884,Z 1169.872,A -85,B 0,C 180,E1 25470.641,E2 25470.641} C_VEL
LIN {X 0,Y 535.905,Z 1169.526,A -85,B 0,C 180,E1 25468.182,E2 25468.182} C_VEL
LIN {X 0,Y 535.917,Z 1167.616,A -85,B 0,C 180,E1 25465.827,E2 25465.827} C_VEL
LIN {X 0,Y 535.922,Z 1164.08,A -85,B 0,C 180,E1 25463.357,E2 25463.357} C_VEL
LIN {X 0,Y 535.972,Z 1159.572,A -85,B 0,C 180,E1 25461.201,E2 25461.201} C_VEL
LIN {X 0,Y 536.051,Z 1153.176,A -85,B 0,C 180,E1 25458.814,E2 25458.814} C_VEL
LIN {X 0,Y 536.197,Z 1145.338,A -85,B 0,C 180,E1 25456.521,E2 25456.521} C_VEL
LIN {X 0,Y 536.468,Z 1135.94,A -85,B 0,C 180,E1 25454.21,E2 25454.21} C_VEL
LIN {X 0,Y 536.841,Z 1125.145,A -85,B 0,C 180,E1 25451.99,E2 25451.99} C_VEL
LIN {X 0,Y 537.394,Z 1111.862,A -85,B 0,C 180,E1 25449.639,E2 25449.639} C_VEL
LIN {X 0,Y 538.013,Z 1098.558,A -85,B 0,C 180,E1 25447.605,E2 25447.605} C_VEL
LIN {X 0,Y 538.864,Z 1082.264,A -85,B 0,C 180,E1 25445.441,E2 25445.441} C_VEL
LIN {X 0,Y 539.84,Z 1065.431,A -85,B 0,C 180,E1 25443.489,E2 25443.489} C_VEL
LIN {X 0,Y 540.865,Z 1047.571,A -85,B 0,C 180,E1 25441.694,E2 25441.694} C_VEL
LIN {X 0,Y 542.074,Z 1027.522,A -85,B 0,C 180,E1 25439.948,E2 25439.948} C_VEL
LIN {X 0,Y 543.282,Z 1007.473,A -85,B 0,C 180,E1 25438.441,E2 25438.441} C_VEL
LIN {X 0,Y 544.416,Z 986.824,A -85,B 0,C 180,E1 25437.131,E2 25437.131} C_VEL
LIN {X 0,Y 545.532,Z 965.202,A -85,B 0,C 180,E1 25435.97,E2 25435.97} C_VEL
LIN {X 0,Y 546.459,Z 945.188,A -85,B 0,C 180,E1 25435.093,E2 25435.093} C_VEL
LIN {X 0,Y 547.35,Z 922.885,A -85,B 0,C 180,E1 25434.301,E2 25434.301} C_VEL
LIN {X 0,Y 547.984,Z 900.821,A -85,B 0,C 180,E1 25433.719,E2 25433.719} C_VEL
LIN {X 0,Y 548.531,Z 872.871,A -85,B 0,C 180,E1 25433.218,E2 25433.218} C_VEL
LIN {X 0,Y 550.656,Z 671.58,A -85,B 0,C 180,E1 25430.108,E2 25430.108} C_VEL
LIN {X 0,Y 551.774,Z 558.036,A -85,B 0,C 180,E1 25428.294,E2 25428.294} C_VEL
LIN {X 0,Y 548.512,Z 542.539,A -85,B 0,C 180,E1 25427.699,E2 25427.699} C_VEL
LIN {X 0,Y 540.183,Z 524.439,A -85,B 0,C 180,E1 25425.448,E2 25425.448} C_VEL
LIN {X 0,Y 536.541,Z 516.988,A -85,B 0,C 180,E1 25424.46,E2 25424.46} C_VEL
LIN {X 0,Y 536.413,Z 516.224,A -85,B 0,C 180,E1 25424.345,E2 25424.345} C_VEL
LIN {X 0,Y 536.422,Z 516.227,A -85,B 0,C 180,E1 25420.82,E2 25420.82} C_VEL
LIN {X 0,Y 536.46,Z 516.224,A -85,B 0,C 180,E1 25417.55,E2 25417.55} C_VEL
LIN {X 0,Y 536.417,Z 516.211,A -85,B 0,C 180,E1 25414.146,E2 25414.146} C_VEL
LIN {X 0,Y 536.466,Z 516.215,A -85,B 0,C 180,E1 25410.771,E2 25410.771} C_VEL
LIN {X 0,Y 536.444,Z 516.219,A -85,B 0,C 180,E1 25407.411,E2 25407.411} C_VEL
LIN {X 0,Y 536.436,Z 516.205,A -85,B 0,C 180,E1 25403.974,E2 25403.974} C_VEL
LIN {X 0,Y 536.46,Z 516.223,A -85,B 0,C 180,E1 25400.625,E2 25400.625} C_VEL
LIN {X 0,Y 536.437,Z 516.203,A -85,B 0,C 180,E1 25397.239,E2 25397.239} C_VEL
LIN {X 0,Y 536.466,Z 516.218,A -85,B 0,C 180,E1 25393.802,E2 25393.802} C_VEL
LIN {X 0,Y 536.454,Z 516.206,A -85,B 0,C 180,E1 25390.307,E2 25390.307} C_VEL
LIN {X 0,Y 536.448,Z 516.223,A -85,B 0,C 180,E1 25386.958,E2 25386.958} C_VEL
LIN {X 0,Y 536.447,Z 516.222,A -85,B 0,C 180,E1 25383.633,E2 25383.633} C_VEL
LIN {X 0,Y 536.464,Z 516.226,A -85,B 0,C 180,E1 25380.213,E2 25380.213} C_VEL
LIN {X 0,Y 536.461,Z 516.22,A -85,B 0,C 180,E1 25376.687,E2 25376.687} C_VEL
LIN {X 0,Y 536.436,Z 516.224,A -85,B 0,C 180,E1 25373.256,E2 25373.256} C_VEL
LIN {X 0,Y 536.459,Z 516.206,A -85,B 0,C 180,E1 25369.91,E2 25369.91} C_VEL
LIN {X 0,Y 536.442,Z 516.221,A -85,B 0,C 180,E1 25366.527,E2 25366.527} C_VEL
LIN {X 0,Y 536.434,Z 516.204,A -85,B 0,C 180,E1 25363.096,E2 25363.096} C_VEL
LIN {X 0,Y 536.464,Z 516.22,A -85,B 0,C 180,E1 25359.716,E2 25359.716} C_VEL
LIN {X 0,Y 536.415,Z 516.204,A -85,B 0,C 180,E1 25356.491,E2 25356.491} C_VEL
LIN {X 0,Y 536.469,Z 516.225,A -85,B 0,C 180,E1 25353.19,E2 25353.19} C_VEL
LIN {X 0,Y 536.411,Z 516.212,A -85,B 0,C 180,E1 25349.907,E2 25349.907} C_VEL
LIN {X 0,Y 536.43,Z 516.218,A -85,B 0,C 180,E1 25346.515,E2 25346.515} C_VEL
LIN {X 0,Y 536.425,Z 516.212,A -85,B 0,C 180,E1 25345.402,E2 25345.402} C_VEL
LIN {X 0,Y 535.476,Z 516.334,A -85,B 0,C 180,E1 25344.579,E2 25344.579} C_VEL
LIN {X 0,Y 528.993,Z 517.151,A -85,B 0,C 180,E1 25342.268,E2 25342.268} C_VEL
LIN {X 0,Y 528.459,Z 517.211,A -85,B 0,C 180,E1 25341.665,E2 25341.665} C_VEL
LIN {X 0,Y 528.505,Z 517.215,A -85,B 0,C 180,E1 25338.357,E2 25338.357} C_VEL
LIN {X 0,Y 528.455,Z 517.222,A -85,B 0,C 180,E1 25335.196,E2 25335.196} C_VEL
LIN {X 0,Y 528.513,Z 517.309,A -85,B 0,C 180,E1 25334.163,E2 25334.163} C_VEL
LIN {X 0,Y 529.709,Z 520.572,A -85,B 0,C 180,E1 25333.976,E2 25333.976} C_VEL
LIN {X 0,Y 532.068,Z 523.418,A -85,B 0,C 180,E1 25333.676,E2 25333.676} C_VEL
LIN {X 0,Y 534.882,Z 527.474,A -85,B 0,C 180,E1 25333.312,E2 25333.312} C_VEL
LIN {X 0,Y 545.738,Z 543.707,A -85,B 0,C 180,E1 25331.956,E2 25331.956} C_VEL
LIN {X 0,Y 543.476,Z 728.775,A -85,B 0,C 180,E1 25329.014,E2 25329.014} C_VEL
LIN {X 0,Y 541.8,Z 862.309,A -85,B 0,C 180,E1 25326.918,E2 25326.918} C_VEL
LIN {X 0,Y 541.069,Z 885.447,A -85,B 0,C 180,E1 25326.369,E2 25326.369} C_VEL
LIN {X 0,Y 540.2,Z 906.873,A -85,B 0,C 180,E1 25325.681,E2 25325.681} C_VEL
LIN {X 0,Y 539.163,Z 928.28,A -85,B 0,C 180,E1 25324.793,E2 25324.793} C_VEL
LIN {X 0,Y 538.102,Z 947.667,A -85,B 0,C 180,E1 25323.821,E2 25323.821} C_VEL
LIN {X 0,Y 536.738,Z 969.496,A -85,B 0,C 180,E1 25322.509,E2 25322.509} C_VEL
LIN {X 0,Y 535.475,Z 989.621,A -85,B 0,C 180,E1 25321.084,E2 25321.084} C_VEL
LIN {X 0,Y 534.097,Z 1009.443,A -85,B 0,C 180,E1 25319.434,E2 25319.434} C_VEL
LIN {X 0,Y 532.803,Z 1028.929,A -85,B 0,C 180,E1 25317.554,E2 25317.554} C_VEL
LIN {X 0,Y 531.717,Z 1045.783,A -85,B 0,C 180,E1 25315.687,E2 25315.687} C_VEL
LIN {X 0,Y 530.713,Z 1061.668,A -85,B 0,C 180,E1 25313.659,E2 25313.659} C_VEL
LIN {X 0,Y 529.885,Z 1076.649,A -85,B 0,C 180,E1 25311.474,E2 25311.474} C_VEL
LIN {X 0,Y 529.238,Z 1089.479,A -85,B 0,C 180,E1 25309.307,E2 25309.307} C_VEL
LIN {X 0,Y 528.707,Z 1101.84,A -85,B 0,C 180,E1 25306.879,E2 25306.879} C_VEL
LIN {X 0,Y 528.366,Z 1111.806,A -85,B 0,C 180,E1 25304.578,E2 25304.578} C_VEL
LIN {X 0,Y 528.116,Z 1120.554,A -85,B 0,C 180,E1 25302.132,E2 25302.132} C_VEL
LIN {X 0,Y 527.983,Z 1127.348,A -85,B 0,C 180,E1 25299.813,E2 25299.813} C_VEL
LIN {X 0,Y 527.922,Z 1132.756,A -85,B 0,C 180,E1 25297.4,E2 25297.4} C_VEL
LIN {X 0,Y 527.912,Z 1136.37,A -85,B 0,C 180,E1 25295.216,E2 25295.216} C_VEL
LIN {X 0,Y 527.899,Z 1138.959,A -85,B 0,C 180,E1 25292.714,E2 25292.714} C_VEL
LIN {X 0,Y 527.887,Z 1139.885,A -85,B 0,C 180,E1 25290.543,E2 25290.543} C_VEL
LIN {X 0,Y 527.908,Z 1139.487,A -85,B 0,C 180,E1 25288.047,E2 25288.047} C_VEL
LIN {X 0,Y 527.914,Z 1137.664,A -85,B 0,C 180,E1 25285.764,E2 25285.764} C_VEL
LIN {X 0,Y 527.919,Z 1134.166,A -85,B 0,C 180,E1 25283.257,E2 25283.257} C_VEL
LIN {X 0,Y 527.983,Z 1129.422,A -85,B 0,C 180,E1 25280.957,E2 25280.957} C_VEL
LIN {X 0,Y 528.088,Z 1122.615,A -85,B 0,C 180,E1 25278.423,E2 25278.423} C_VEL
LIN {X 0,Y 528.255,Z 1114.955,A -85,B 0,C 180,E1 25276.164,E2 25276.164} C_VEL
LIN {X 0,Y 528.577,Z 1105.115,A -85,B 0,C 180,E1 25273.742,E2 25273.742} C_VEL
LIN {X 0,Y 528.982,Z 1094.782,A -85,B 0,C 180,E1 25271.597,E2 25271.597} C_VEL
LIN {X 0,Y 529.621,Z 1081.435,A -85,B 0,C 180,E1 25269.212,E2 25269.212} C_VEL
LIN {X 0,Y 530.4,Z 1067.306,A -85,B 0,C 180,E1 25267.032,E2 25267.032} C_VEL
LIN {X 0,Y 531.32,Z 1051.691,A -85,B 0,C 180,E1 25264.95,E2 25264.95} C_VEL
LIN {X 0,Y 532.427,Z 1034.743,A -85,B 0,C 180,E1 25262.97,E2 25262.97} C_VEL
LIN {X 0,Y 533.574,Z 1017.415,A -85,B 0,C 180,E1 25261.211,E2 25261.211} C_VEL
LIN {X 0,Y 534.917,Z 997.335,A -85,B 0,C 180,E1 25259.442,E2 25259.442} C_VEL
LIN {X 0,Y 536.304,Z 977.033,A -85,B 0,C 180,E1 25257.904,E2 25257.904} C_VEL
LIN {X 0,Y 537.545,Z 956.531,A -85,B 0,C 180,E1 25256.594,E2 25256.594} C_VEL
LIN {X 0,Y 538.845,Z 934.406,A -85,B 0,C 180,E1 25255.403,E2 25255.403} C_VEL
LIN {X 0,Y 539.846,Z 914.741,A -85,B 0,C 180,E1 25254.537,E2 25254.537} C_VEL
LIN {X 0,Y 540.816,Z 892.379,A -85,B 0,C 180,E1 25253.741,E2 25253.741} C_VEL
LIN {X 0,Y 541.534,Z 870.663,A -85,B 0,C 180,E1 25253.167,E2 25253.167} C_VEL
LIN {X 0,Y 542.137,Z 841.98,A -85,B 0,C 180,E1 25252.652,E2 25252.652} C_VEL
LIN {X 0,Y 544.591,Z 636.757,A -85,B 0,C 180,E1 25249.446,E2 25249.446} C_VEL
LIN {X 0,Y 545.626,Z 543.355,A -85,B 0,C 180,E1 25247.938,E2 25247.938} C_VEL
LIN {X 0,Y 534.598,Z 527.212,A -85,B 0,C 180,E1 25246.564,E2 25246.564} C_VEL
LIN {X 0,Y 531.969,Z 523.232,A -85,B 0,C 180,E1 25246.22,E2 25246.22} C_VEL
LIN {X 0,Y 529.138,Z 519.534,A -85,B 0,C 180,E1 25245.855,E2 25245.855} C_VEL
LIN {X 0,Y 528.502,Z 517.219,A -85,B 0,C 180,E1 25245.725,E2 25245.725} C_VEL
LIN {X 0,Y 528.447,Z 517.22,A -85,B 0,C 180,E1 25242.446,E2 25242.446} C_VEL
LIN {X 0,Y 528.521,Z 517.196,A -85,B 0,C 180,E1 25239.188,E2 25239.188} C_VEL
LIN {X 0,Y 528.46,Z 517.217,A -85,B 0,C 180,E1 25235.911,E2 25235.911} C_VEL
LIN {X 0,Y 528.484,Z 517.216,A -85,B 0,C 180,E1 25232.456,E2 25232.456} C_VEL
LIN {X 0,Y 528.488,Z 517.197,A -85,B 0,C 180,E1 25229.287,E2 25229.287} C_VEL
LIN {X 0,Y 528.478,Z 517.214,A -85,B 0,C 180,E1 25225.916,E2 25225.916} C_VEL
LIN {X 0,Y 528.526,Z 517.195,A -85,B 0,C 180,E1 25222.584,E2 25222.584} C_VEL
LIN {X 0,Y 528.481,Z 517.214,A -85,B 0,C 180,E1 25219.22,E2 25219.22} C_VEL
LIN {X 0,Y 528.518,Z 517.203,A -85,B 0,C 180,E1 25215.809,E2 25215.809} C_VEL
LIN {X 0,Y 528.522,Z 517.211,A -85,B 0,C 180,E1 25212.344,E2 25212.344} C_VEL
LIN {X 0,Y 528.492,Z 517.211,A -85,B 0,C 180,E1 25208.925,E2 25208.925} C_VEL
LIN {X 0,Y 528.52,Z 517.206,A -85,B 0,C 180,E1 25205.537,E2 25205.537} C_VEL
LIN {X 0,Y 528.518,Z 517.214,A -85,B 0,C 180,E1 25202.06,E2 25202.06} C_VEL
LIN {X 0,Y 528.507,Z 517.21,A -85,B 0,C 180,E1 25198.591,E2 25198.591} C_VEL
LIN {X 0,Y 528.513,Z 517.21,A -85,B 0,C 180,E1 25195.225,E2 25195.225} C_VEL
LIN {X 0,Y 528.513,Z 517.214,A -85,B 0,C 180,E1 25191.843,E2 25191.843} C_VEL
LIN {X 0,Y 528.519,Z 517.188,A -85,B 0,C 180,E1 25188.322,E2 25188.322} C_VEL
LIN {X 0,Y 528.505,Z 517.211,A -85,B 0,C 180,E1 25184.866,E2 25184.866} C_VEL
LIN {X 0,Y 528.517,Z 517.193,A -85,B 0,C 180,E1 25181.406,E2 25181.406} C_VEL
LIN {X 0,Y 528.512,Z 517.208,A -85,B 0,C 180,E1 25177.972,E2 25177.972} C_VEL
LIN {X 0,Y 528.497,Z 517.216,A -85,B 0,C 180,E1 25174.447,E2 25174.447} C_VEL
LIN {X 0,Y 528.524,Z 517.196,A -85,B 0,C 180,E1 25171.034,E2 25171.034} C_VEL
LIN {X 0,Y 528.487,Z 517.212,A -85,B 0,C 180,E1 25167.746,E2 25167.746} C_VEL
LIN {X 0,Y 528.501,Z 517.216,A -85,B 0,C 180,E1 25164.254,E2 25164.254} C_VEL
LIN {X 0,Y 528.519,Z 517.201,A -85,B 0,C 180,E1 25160.863,E2 25160.863} C_VEL
LIN {X 0,Y 528.471,Z 517.204,A -85,B 0,C 180,E1 25157.512,E2 25157.512} C_VEL
LIN {X 0,Y 528.553,Z 517.4,A -85,B 0,C 180,E1 25156.359,E2 25156.359} C_VEL
LIN {X 0,Y 529.596,Z 520.367,A -85,B 0,C 180,E1 25155.992,E2 25155.992} C_VEL
LIN {X 0,Y 530.785,Z 522.723,A -85,B 0,C 180,E1 25155.664,E2 25155.664} C_VEL
LIN {X 0,Y 539.828,Z 541.491,A -85,B 0,C 180,E1 25153.212,E2 25153.212} C_VEL
LIN {X 0,Y 541.098,Z 543.973,A -85,B 0,C 180,E1 25152.968,E2 25152.968} C_VEL
LIN {X 0,Y 543.259,Z 547.867,A -85,B 0,C 180,E1 25152.69,E2 25152.69} C_VEL
LIN {X 0,Y 545.932,Z 561.598,A -85,B 0,C 180,E1 25152.193,E2 25152.193} C_VEL
LIN {X 0,Y 543.64,Z 743.608,A -85,B 0,C 180,E1 25149.298,E2 25149.298} C_VEL
LIN {X 0,Y 541.804,Z 892.156,A -85,B 0,C 180,E1 25146.965,E2 25146.965} C_VEL
LIN {X 0,Y 541.078,Z 915.228,A -85,B 0,C 180,E1 25146.42,E2 25146.42} C_VEL
LIN {X 0,Y 540.209,Z 936.566,A -85,B 0,C 180,E1 25145.737,E2 25145.737} C_VEL
LIN {X 0,Y 539.16,Z 958.393,A -85,B 0,C 180,E1 25144.832,E2 25144.832} C_VEL
LIN {X 0,Y 538.07,Z 978.214,A -85,B 0,C 180,E1 25143.837,E2 25143.837} C_VEL
LIN {X 0,Y 536.752,Z 999.244,A -85,B 0,C 180,E1 25142.571,E2 25142.571} C_VEL
LIN {X 0,Y 535.49,Z 1019.409,A -85,B 0,C 180,E1 25141.145,E2 25141.145} C_VEL
LIN {X 0,Y 534.109,Z 1039.274,A -85,B 0,C 180,E1 25139.494,E2 25139.494} C_VEL
LIN {X 0,Y 532.815,Z 1058.791,A -85,B 0,C 180,E1 25137.614,E2 25137.614} C_VEL
LIN {X 0,Y 531.724,Z 1075.661,A -85,B 0,C 180,E1 25135.745,E2 25135.745} C_VEL
LIN {X 0,Y 530.695,Z 1091.995,A -85,B 0,C 180,E1 25133.66,E2 25133.66} C_VEL
LIN {X 0,Y 529.867,Z 1106.926,A -85,B 0,C 180,E1 25131.474,E2 25131.474} C_VEL
LIN {X 0,Y 529.228,Z 1119.73,A -85,B 0,C 180,E1 25129.306,E2 25129.306} C_VEL
LIN {X 0,Y 528.698,Z 1132.052,A -85,B 0,C 180,E1 25126.878,E2 25126.878} C_VEL
LIN {X 0,Y 528.362,Z 1141.991,A -85,B 0,C 180,E1 25124.577,E2 25124.577} C_VEL
LIN {X 0,Y 528.118,Z 1150.701,A -85,B 0,C 180,E1 25122.131,E2 25122.131} C_VEL
LIN {X 0,Y 527.982,Z 1157.474,A -85,B 0,C 180,E1 25119.813,E2 25119.813} C_VEL
LIN {X 0,Y 527.919,Z 1162.841,A -85,B 0,C 180,E1 25117.399,E2 25117.399} C_VEL
LIN {X 0,Y 527.914,Z 1166.437,A -85,B 0,C 180,E1 25115.216,E2 25115.216} C_VEL
LIN {X 0,Y 527.909,Z 1169.056,A -85,B 0,C 180,E1 25112.605,E2 25112.605} C_VEL
LIN {X 0,Y 527.891,Z 1169.939,A -85,B 0,C 180,E1 25110.325,E2 25110.325} C_VEL
LIN {X 0,Y 527.914,Z 1169.324,A -85,B 0,C 180,E1 25107.829,E2 25107.829} C_VEL
LIN {X 0,Y 527.909,Z 1167.389,A -85,B 0,C 180,E1 25105.546,E2 25105.546} C_VEL
LIN {X 0,Y 527.911,Z 1163.667,A -85,B 0,C 180,E1 25103.037,E2 25103.037} C_VEL
LIN {X 0,Y 527.985,Z 1159.062,A -85,B 0,C 180,E1 25100.847,E2 25100.847} C_VEL
LIN {X 0,Y 528.101,Z 1152.116,A -85,B 0,C 180,E1 25098.312,E2 25098.312} C_VEL
LIN {X 0,Y 528.269,Z 1144.521,A -85,B 0,C 180,E1 25096.091,E2 25096.091} C_VEL
LIN {X 0,Y 528.602,Z 1134.395,A -85,B 0,C 180,E1 25093.63,E2 25093.63} C_VEL
LIN {X 0,Y 529.043,Z 1123.405,A -85,B 0,C 180,E1 25091.373,E2 25091.373} C_VEL
LIN {X 0,Y 529.663,Z 1110.459,A -85,B 0,C 180,E1 25089.097,E2 25089.097} C_VEL
LIN {X 0,Y 530.476,Z 1096.055,A -85,B 0,C 180,E1 25086.895,E2 25086.895} C_VEL
LIN {X 0,Y 531.415,Z 1080.31,A -85,B 0,C 180,E1 25084.823,E2 25084.823} C_VEL
LIN {X 0,Y 532.574,Z 1062.114,A -85,B 0,C 180,E1 25082.736,E2 25082.736} C_VEL
LIN {X 0,Y 533.839,Z 1043.896,A -85,B 0,C 180,E1 25080.919,E2 25080.919} C_VEL
LIN {X 0,Y 535.099,Z 1024.558,A -85,B 0,C 180,E1 25079.263,E2 25079.263} C_VEL
LIN {X 0,Y 536.494,Z 1003.721,A -85,B 0,C 180,E1 25077.727,E2 25077.727} C_VEL
LIN {X 0,Y 537.71,Z 983.806,A -85,B 0,C 180,E1 25076.477,E2 25076.477} C_VEL
LIN {X 0,Y 538.96,Z 962.235,A -85,B 0,C 180,E1 25075.346,E2 25075.346} C_VEL
LIN {X 0,Y 539.935,Z 942.966,A -85,B 0,C 180,E1 25074.511,E2 25074.511} C_VEL
LIN {X 0,Y 540.911,Z 919.195,A -85,B 0,C 180,E1 25073.692,E2 25073.692} C_VEL
LIN {X 0,Y 541.654,Z 897.736,A -85,B 0,C 180,E1 25073.147,E2 25073.147} C_VEL
LIN {X 0,Y 542.21,Z 865.364,A -85,B 0,C 180,E1 25072.595,E2 25072.595} C_VEL
LIN {X 0,Y 544.652,Z 662.037,A -85,B 0,C 180,E1 25069.416,E2 25069.416} C_VEL
LIN {X 0,Y 545.775,Z 559.806,A -85,B 0,C 180,E1 25067.761,E2 25067.761} C_VEL
LIN {X 0,Y 542.883,Z 546.838,A -85,B 0,C 180,E1 25067.256,E2 25067.256} C_VEL
LIN {X 0,Y 540.231,Z 542.479,A -85,B 0,C 180,E1 25066.905,E2 25066.905} C_VEL
LIN {X 0,Y 531.977,Z 525.112,A -85,B 0,C 180,E1 25064.663,E2 25064.663} C_VEL
LIN {X 0,Y 528.769,Z 518.417,A -85,B 0,C 180,E1 25063.752,E2 25063.752} C_VEL
LIN {X 0,Y 528.529,Z 517.214,A -85,B 0,C 180,E1 25063.618,E2 25063.618} C_VEL
LIN {X 0,Y 528.475,Z 517.219,A -85,B 0,C 180,E1 25060.317,E2 25060.317} C_VEL
LIN {X 0,Y 528.516,Z 517.214,A -85,B 0,C 180,E1 25056.984,E2 25056.984} C_VEL
LIN {X 0,Y 528.5,Z 517.198,A -85,B 0,C 180,E1 25053.65,E2 25053.65} C_VEL
LIN {X 0,Y 528.488,Z 517.206,A -85,B 0,C 180,E1 25050.215,E2 25050.215} C_VEL
LIN {X 0,Y 528.524,Z 517.212,A -85,B 0,C 180,E1 25046.881,E2 25046.881} C_VEL
LIN {X 0,Y 528.493,Z 517.191,A -85,B 0,C 180,E1 25043.527,E2 25043.527} C_VEL
LIN {X 0,Y 528.522,Z 517.206,A -85,B 0,C 180,E1 25040.139,E2 25040.139} C_VEL
LIN {X 0,Y 528.52,Z 517.195,A -85,B 0,C 180,E1 25036.598,E2 25036.598} C_VEL
LIN {X 0,Y 528.504,Z 517.212,A -85,B 0,C 180,E1 25033.233,E2 25033.233} C_VEL
LIN {X 0,Y 528.515,Z 517.2,A -85,B 0,C 180,E1 25029.803,E2 25029.803} C_VEL
LIN {X 0,Y 528.522,Z 517.211,A -85,B 0,C 180,E1 25026.299,E2 25026.299} C_VEL
LIN {X 0,Y 528.513,Z 517.211,A -85,B 0,C 180,E1 25022.819,E2 25022.819} C_VEL
LIN {X 0,Y 528.505,Z 517.21,A -85,B 0,C 180,E1 25019.458,E2 25019.458} C_VEL
LIN {X 0,Y 528.522,Z 517.215,A -85,B 0,C 180,E1 25015.986,E2 25015.986} C_VEL
LIN {X 0,Y 528.524,Z 517.21,A -85,B 0,C 180,E1 25012.442,E2 25012.442} C_VEL
LIN {X 0,Y 528.491,Z 517.193,A -85,B 0,C 180,E1 25009.086,E2 25009.086} C_VEL
LIN {X 0,Y 528.528,Z 517.215,A -85,B 0,C 180,E1 25005.651,E2 25005.651} C_VEL
LIN {X 0,Y 528.5,Z 517.187,A -85,B 0,C 180,E1 25002.266,E2 25002.266} C_VEL
LIN {X 0,Y 528.488,Z 517.214,A -85,B 0,C 180,E1 24998.816,E2 24998.816} C_VEL
LIN {X 0,Y 528.524,Z 517.189,A -85,B 0,C 180,E1 24995.5,E2 24995.5} C_VEL
LIN {X 0,Y 528.474,Z 517.211,A -85,B 0,C 180,E1 24992.14,E2 24992.14} C_VEL
LIN {X 0,Y 528.51,Z 517.209,A -85,B 0,C 180,E1 24988.773,E2 24988.773} C_VEL
LIN {X 0,Y 528.476,Z 517.201,A -85,B 0,C 180,E1 24985.549,E2 24985.549} C_VEL
LIN {X 0,Y 528.467,Z 517.212,A -85,B 0,C 180,E1 24982.055,E2 24982.055} C_VEL
LIN {X 0,Y 528.459,Z 517.211,A -85,B 0,C 180,E1 24981.665,E2 24981.665} C_VEL
LIN {X 0,Y 527.489,Z 517.333,A -85,B 0,C 180,E1 24980.83,E2 24980.83} C_VEL
LIN {X 0,Y 520.984,Z 518.153,A -85,B 0,C 180,E1 24978.423,E2 24978.423} C_VEL
LIN {X 0,Y 520.523,Z 518.206,A -85,B 0,C 180,E1 24977.872,E2 24977.872} C_VEL
LIN {X 0,Y 520.544,Z 518.343,A -85,B 0,C 180,E1 24975.011,E2 24975.011} C_VEL
LIN {X 0,Y 521.801,Z 521.621,A -85,B 0,C 180,E1 24974.809,E2 24974.809} C_VEL
LIN {X 0,Y 524.216,Z 524.381,A -85,B 0,C 180,E1 24974.492,E2 24974.492} C_VEL
LIN {X 0,Y 526.898,Z 528.368,A -85,B 0,C 180,E1 24974.128,E2 24974.128} C_VEL
LIN {X 0,Y 537.755,Z 544.199,A -85,B 0,C 180,E1 24972.721,E2 24972.721} C_VEL
LIN {X 0,Y 539.748,Z 547.402,A -85,B 0,C 180,E1 24972.467,E2 24972.467} C_VEL
LIN {X 0,Y 537.213,Z 732.576,A -85,B 0,C 180,E1 24969.493,E2 24969.493} C_VEL
LIN {X 0,Y 535.4,Z 862.46,A -85,B 0,C 180,E1 24967.432,E2 24967.432} C_VEL
LIN {X 0,Y 534.609,Z 885.364,A -85,B 0,C 180,E1 24966.884,E2 24966.884} C_VEL
LIN {X 0,Y 533.667,Z 906.467,A -85,B 0,C 180,E1 24966.203,E2 24966.203} C_VEL
LIN {X 0,Y 532.496,Z 928.208,A -85,B 0,C 180,E1 24965.297,E2 24965.297} C_VEL
LIN {X 0,Y 531.257,Z 948.915,A -85,B 0,C 180,E1 24964.246,E2 24964.246} C_VEL
LIN {X 0,Y 529.752,Z 970.404,A -85,B 0,C 180,E1 24962.928,E2 24962.928} C_VEL
LIN {X 0,Y 528.353,Z 990.391,A -85,B 0,C 180,E1 24961.487,E2 24961.487} C_VEL
LIN {X 0,Y 526.862,Z 1009.696,A -85,B 0,C 180,E1 24959.856,E2 24959.856} C_VEL
LIN {X 0,Y 525.394,Z 1029.49,A -85,B 0,C 180,E1 24957.915,E2 24957.915} C_VEL
LIN {X 0,Y 524.15,Z 1046.796,A -85,B 0,C 180,E1 24955.963,E2 24955.963} C_VEL
LIN {X 0,Y 523.034,Z 1062.517,A -85,B 0,C 180,E1 24953.908,E2 24953.908} C_VEL
LIN {X 0,Y 522.062,Z 1078.072,A -85,B 0,C 180,E1 24951.576,E2 24951.576} C_VEL
LIN {X 0,Y 521.332,Z 1091.386,A -85,B 0,C 180,E1 24949.262,E2 24949.262} C_VEL
LIN {X 0,Y 520.764,Z 1103.163,A -85,B 0,C 180,E1 24946.853,E2 24946.853} C_VEL
LIN {X 0,Y 520.373,Z 1113.542,A -85,B 0,C 180,E1 24944.351,E2 24944.351} C_VEL
LIN {X 0,Y 520.134,Z 1121.268,A -85,B 0,C 180,E1 24942.095,E2 24942.095} C_VEL
LIN {X 0,Y 519.986,Z 1128.194,A -85,B 0,C 180,E1 24939.631,E2 24939.631} C_VEL
LIN {X 0,Y 519.918,Z 1133.17,A -85,B 0,C 180,E1 24937.292,E2 24937.292} C_VEL
LIN {X 0,Y 519.913,Z 1136.998,A -85,B 0,C 180,E1 24934.854,E2 24934.854} C_VEL
LIN {X 0,Y 519.915,Z 1139.23,A -85,B 0,C 180,E1 24932.315,E2 24932.315} C_VEL
LIN {X 0,Y 519.899,Z 1139.971,A -85,B 0,C 180,E1 24929.78,E2 24929.78} C_VEL
LIN {X 0,Y 519.912,Z 1139.151,A -85,B 0,C 180,E1 24927.465,E2 24927.465} C_VEL
LIN {X 0,Y 519.914,Z 1136.82,A -85,B 0,C 180,E1 24924.925,E2 24924.925} C_VEL
LIN {X 0,Y 519.918,Z 1133.132,A -85,B 0,C 180,E1 24922.597,E2 24922.597} C_VEL
LIN {X 0,Y 519.987,Z 1128.145,A -85,B 0,C 180,E1 24920.258,E2 24920.258} C_VEL
LIN {X 0,Y 520.139,Z 1121.199,A -85,B 0,C 180,E1 24917.793,E2 24917.793} C_VEL
LIN {X 0,Y 520.395,Z 1113.049,A -85,B 0,C 180,E1 24915.422,E2 24915.422} C_VEL
LIN {X 0,Y 520.782,Z 1102.738,A -85,B 0,C 180,E1 24912.964,E2 24912.964} C_VEL
LIN {X 0,Y 521.34,Z 1091.243,A -85,B 0,C 180,E1 24910.623,E2 24910.623} C_VEL
LIN {X 0,Y 522.026,Z 1078.616,A -85,B 0,C 180,E1 24908.423,E2 24908.423} C_VEL
LIN {X 0,Y 522.991,Z 1063.155,A -85,B 0,C 180,E1 24906.09,E2 24906.09} C_VEL
LIN {X 0,Y 524.144,Z 1046.9,A -85,B 0,C 180,E1 24903.959,E2 24903.959} C_VEL
LIN {X 0,Y 525.385,Z 1029.639,A -85,B 0,C 180,E1 24902.011,E2 24902.011} C_VEL
LIN {X 0,Y 526.824,Z 1010.242,A -85,B 0,C 180,E1 24900.103,E2 24900.103} C_VEL
LIN {X 0,Y 528.268,Z 991.443,A -85,B 0,C 180,E1 24898.507,E2 24898.507} C_VEL
LIN {X 0,Y 529.729,Z 970.77,A -85,B 0,C 180,E1 24897.007,E2 24897.007} C_VEL
LIN {X 0,Y 531.229,Z 949.346,A -85,B 0,C 180,E1 24895.688,E2 24895.688} C_VEL
LIN {X 0,Y 532.441,Z 929.266,A -85,B 0,C 180,E1 24894.663,E2 24894.663} C_VEL
LIN {X 0,Y 533.629,Z 907.303,A -85,B 0,C 180,E1 24893.736,E2 24893.736} C_VEL
LIN {X 0,Y 534.589,Z 885.842,A -85,B 0,C 180,E1 24893.04,E2 24893.04} C_VEL
LIN {X 0,Y 535.396,Z 862.887,A -85,B 0,C 180,E1 24892.486,E2 24892.486} C_VEL
LIN {X 0,Y 536.763,Z 766.413,A -85,B 0,C 180,E1 24890.95,E2 24890.95} C_VEL
LIN {X 0,Y 539.473,Z 566.572,A -85,B 0,C 180,E1 24887.756,E2 24887.756} C_VEL
LIN {X 0,Y 539.598,Z 546.895,A -85,B 0,C 180,E1 24887.419,E2 24887.419} C_VEL
LIN {X 0,Y 529.729,Z 532.559,A -85,B 0,C 180,E1 24886.158,E2 24886.158} C_VEL
LIN {X 0,Y 526.458,Z 527.908,A -85,B 0,C 180,E1 24885.726,E2 24885.726} C_VEL
LIN {X 0,Y 523.466,Z 523.444,A -85,B 0,C 180,E1 24885.319,E2 24885.319} C_VEL
LIN {X 0,Y 521.235,Z 520.65,A -85,B 0,C 180,E1 24885.02,E2 24885.02} C_VEL
LIN {X 0,Y 520.515,Z 518.212,A -85,B 0,C 180,E1 24884.879,E2 24884.879} C_VEL
LIN {X 0,Y 520.554,Z 518.204,A -85,B 0,C 180,E1 24881.65,E2 24881.65} C_VEL
LIN {X 0,Y 520.515,Z 518.197,A -85,B 0,C 180,E1 24878.349,E2 24878.349} C_VEL
LIN {X 0,Y 520.582,Z 518.182,A -85,B 0,C 180,E1 24875.049,E2 24875.049} C_VEL
LIN {X 0,Y 520.527,Z 518.207,A -85,B 0,C 180,E1 24871.757,E2 24871.757} C_VEL
LIN {X 0,Y 520.554,Z 518.193,A -85,B 0,C 180,E1 24868.322,E2 24868.322} C_VEL
LIN {X 0,Y 520.553,Z 518.198,A -85,B 0,C 180,E1 24865.118,E2 24865.118} C_VEL
LIN {X 0,Y 520.541,Z 518.198,A -85,B 0,C 180,E1 24861.616,E2 24861.616} C_VEL
LIN {X 0,Y 520.588,Z 518.181,A -85,B 0,C 180,E1 24858.244,E2 24858.244} C_VEL
LIN {X 0,Y 520.555,Z 518.197,A -85,B 0,C 180,E1 24854.801,E2 24854.801} C_VEL
LIN {X 0,Y 520.561,Z 518.197,A -85,B 0,C 180,E1 24851.298,E2 24851.298} C_VEL
LIN {X 0,Y 520.584,Z 518.199,A -85,B 0,C 180,E1 24847.949,E2 24847.949} C_VEL
LIN {X 0,Y 520.559,Z 518.198,A -85,B 0,C 180,E1 24844.517,E2 24844.517} C_VEL
LIN {X 0,Y 520.583,Z 518.191,A -85,B 0,C 180,E1 24840.991,E2 24840.991} C_VEL
LIN {X 0,Y 520.577,Z 518.198,A -85,B 0,C 180,E1 24837.468,E2 24837.468} C_VEL
LIN {X 0,Y 520.569,Z 518.199,A -85,B 0,C 180,E1 24834.047,E2 24834.047} C_VEL
LIN {X 0,Y 520.579,Z 518.191,A -85,B 0,C 180,E1 24830.604,E2 24830.604} C_VEL
LIN {X 0,Y 520.573,Z 518.193,A -85,B 0,C 180,E1 24827.127,E2 24827.127} C_VEL
LIN {X 0,Y 520.578,Z 518.195,A -85,B 0,C 180,E1 24823.715,E2 24823.715} C_VEL
LIN {X 0,Y 520.563,Z 518.2,A -85,B 0,C 180,E1 24820.359,E2 24820.359} C_VEL
LIN {X 0,Y 520.579,Z 518.183,A -85,B 0,C 180,E1 24816.926,E2 24816.926} C_VEL
LIN {X 0,Y 520.585,Z 518.2,A -85,B 0,C 180,E1 24813.416,E2 24813.416} C_VEL
LIN {X 0,Y 520.546,Z 518.193,A -85,B 0,C 180,E1 24810.029,E2 24810.029} C_VEL
LIN {X 0,Y 520.583,Z 518.186,A -85,B 0,C 180,E1 24806.666,E2 24806.666} C_VEL
LIN {X 0,Y 520.554,Z 518.203,A -85,B 0,C 180,E1 24803.32,E2 24803.32} C_VEL
LIN {X 0,Y 520.542,Z 518.208,A -85,B 0,C 180,E1 24799.806,E2 24799.806} C_VEL
LIN {X 0,Y 520.566,Z 518.406,A -85,B 0,C 180,E1 24797.162,E2 24797.162} C_VEL
LIN {X 0,Y 521.966,Z 521.81,A -85,B 0,C 180,E1 24796.704,E2 24796.704} C_VEL
LIN {X 0,Y 530.366,Z 539.297,A -85,B 0,C 180,E1 24794.321,E2 24794.321} C_VEL
LIN {X 0,Y 532.318,Z 543.102,A -85,B 0,C 180,E1 24793.862,E2 24793.862} C_VEL
LIN {X 0,Y 537.81,Z 552.026,A -85,B 0,C 180,E1 24793.148,E2 24793.148} C_VEL
LIN {X 0,Y 539.97,Z 563.339,A -85,B 0,C 180,E1 24792.736,E2 24792.736} C_VEL
LIN {X 0,Y 537.423,Z 745.669,A -85,B 0,C 180,E1 24789.807,E2 24789.807} C_VEL
LIN {X 0,Y 535.407,Z 892.185,A -85,B 0,C 180,E1 24787.482,E2 24787.482} C_VEL
LIN {X 0,Y 534.623,Z 915.096,A -85,B 0,C 180,E1 24786.936,E2 24786.936} C_VEL
LIN {X 0,Y 533.694,Z 935.923,A -85,B 0,C 180,E1 24786.267,E2 24786.267} C_VEL
LIN {X 0,Y 532.488,Z 958.39,A -85,B 0,C 180,E1 24785.333,E2 24785.333} C_VEL
LIN {X 0,Y 531.275,Z 978.575,A -85,B 0,C 180,E1 24784.309,E2 24784.309} C_VEL
LIN {X 0,Y 529.77,Z 1000.141,A -85,B 0,C 180,E1 24782.99,E2 24782.99} C_VEL
LIN {X 0,Y 528.372,Z 1020.187,A -85,B 0,C 180,E1 24781.549,E2 24781.549} C_VEL
LIN {X 0,Y 526.893,Z 1039.272,A -85,B 0,C 180,E1 24779.939,E2 24779.939} C_VEL
LIN {X 0,Y 525.422,Z 1059.136,A -85,B 0,C 180,E1 24777.998,E2 24777.998} C_VEL
LIN {X 0,Y 524.212,Z 1075.661,A -85,B 0,C 180,E1 24776.142,E2 24776.142} C_VEL
LIN {X 0,Y 523.068,Z 1091.993,A -85,B 0,C 180,E1 24774.026,E2 24774.026} C_VEL
LIN {X 0,Y 522.118,Z 1107.244,A -85,B 0,C 180,E1 24771.756,E2 24771.756} C_VEL
LIN {X 0,Y 521.408,Z 1119.728,A -85,B 0,C 180,E1 24769.608,E2 24769.608} C_VEL
LIN {X 0,Y 520.821,Z 1131.805,A -85,B 0,C 180,E1 24767.196,E2 24767.196} C_VEL
LIN {X 0,Y 520.439,Z 1141.577,A -85,B 0,C 180,E1 24764.907,E2 24764.907} C_VEL
LIN {X 0,Y 520.155,Z 1150.345,A -85,B 0,C 180,E1 24762.432,E2 24762.432} C_VEL
LIN {X 0,Y 520.017,Z 1156.868,A -85,B 0,C 180,E1 24760.189,E2 24760.189} C_VEL
LIN {X 0,Y 519.939,Z 1162.635,A -85,B 0,C 180,E1 24757.625,E2 24757.625} C_VEL
LIN {X 0,Y 519.908,Z 1166.278,A -85,B 0,C 180,E1 24755.407,E2 24755.407} C_VEL
LIN {X 0,Y 519.893,Z 1168.919,A -85,B 0,C 180,E1 24752.866,E2 24752.866} C_VEL
LIN {X 0,Y 519.884,Z 1169.872,A -85,B 0,C 180,E1 24750.661,E2 24750.661} C_VEL
LIN {X 0,Y 519.906,Z 1169.526,A -85,B 0,C 180,E1 24748.126,E2 24748.126} C_VEL
LIN {X 0,Y 519.914,Z 1167.616,A -85,B 0,C 180,E1 24745.698,E2 24745.698} C_VEL
LIN {X 0,Y 519.918,Z 1164.08,A -85,B 0,C 180,E1 24743.152,E2 24743.152} C_VEL
LIN {X 0,Y 519.991,Z 1159.572,A -85,B 0,C 180,E1 24740.928,E2 24740.928} C_VEL
LIN {X 0,Y 520.104,Z 1153.175,A -85,B 0,C 180,E1 24738.467,E2 24738.467} C_VEL
LIN {X 0,Y 520.298,Z 1145.341,A -85,B 0,C 180,E1 24736.101,E2 24736.101} C_VEL
LIN {X 0,Y 520.644,Z 1135.938,A -85,B 0,C 180,E1 24733.717,E2 24733.717} C_VEL
LIN {X 0,Y 521.118,Z 1125.058,A -85,B 0,C 180,E1 24731.409,E2 24731.409} C_VEL
LIN {X 0,Y 521.83,Z 1111.858,A -85,B 0,C 180,E1 24729.004,E2 24729.004} C_VEL
LIN {X 0,Y 522.649,Z 1098.561,A -85,B 0,C 180,E1 24726.91,E2 24726.91} C_VEL
LIN {X 0,Y 523.704,Z 1082.724,A -85,B 0,C 180,E1 24724.741,E2 24724.741} C_VEL
LIN {X 0,Y 524.928,Z 1065.978,A -85,B 0,C 180,E1 24722.735,E2 24722.735} C_VEL
LIN {X 0,Y 526.238,Z 1048.175,A -85,B 0,C 180,E1 24720.895,E2 24720.895} C_VEL
LIN {X 0,Y 527.725,Z 1028.254,A -85,B 0,C 180,E1 24719.105,E2 24719.105} C_VEL
LIN {X 0,Y 529.163,Z 1009.145,A -85,B 0,C 180,E1 24717.629,E2 24717.629} C_VEL
LIN {X 0,Y 530.627,Z 987.822,A -85,B 0,C 180,E1 24716.229,E2 24716.229} C_VEL
LIN {X 0,Y 532.062,Z 966.057,A -85,B 0,C 180,E1 24715.029,E2 24715.029} C_VEL
LIN {X 0,Y 533.224,Z 945.313,A -85,B 0,C 180,E1 24714.1,E2 24714.1} C_VEL
LIN {X 0,Y 534.286,Z 923.667,A -85,B 0,C 180,E1 24713.312,E2 24713.312} C_VEL
LIN {X 0,Y 535.095,Z 901.307,A -85,B 0,C 180,E1 24712.711,E2 24712.711} C_VEL
LIN {X 0,Y 535.735,Z 875.161,A -85,B 0,C 180,E1 24712.226,E2 24712.226} C_VEL
LIN {X 0,Y 538.392,Z 674.273,A -85,B 0,C 180,E1 24709.055,E2 24709.055} C_VEL
LIN {X 0,Y 539.84,Z 561.791,A -85,B 0,C 180,E1 24707.224,E2 24707.224} C_VEL
LIN {X 0,Y 537.468,Z 551.18,A -85,B 0,C 180,E1 24706.803,E2 24706.803} C_VEL
LIN {X 0,Y 531.773,Z 542.268,A -85,B 0,C 180,E1 24706.065,E2 24706.065} C_VEL
LIN {X 0,Y 523.703,Z 525.458,A -85,B 0,C 180,E1 24703.806,E2 24703.806} C_VEL
LIN {X 0,Y 521.965,Z 521.812,A -85,B 0,C 180,E1 24703.296,E2 24703.296} C_VEL
LIN {X 0,Y 520.565,Z 518.409,A -85,B 0,C 180,E1 24702.838,E2 24702.838} C_VEL
LIN {X 0,Y 520.573,Z 518.203,A -85,B 0,C 180,E1 24699.761,E2 24699.761} C_VEL
LIN {X 0,Y 520.542,Z 518.206,A -85,B 0,C 180,E1 24696.407,E2 24696.407} C_VEL
LIN {X 0,Y 520.587,Z 518.191,A -85,B 0,C 180,E1 24693.056,E2 24693.056} C_VEL
LIN {X 0,Y 520.55,Z 518.186,A -85,B 0,C 180,E1 24689.706,E2 24689.706} C_VEL
LIN {X 0,Y 520.567,Z 518.198,A -85,B 0,C 180,E1 24686.216,E2 24686.216} C_VEL
LIN {X 0,Y 520.583,Z 518.182,A -85,B 0,C 180,E1 24682.791,E2 24682.791} C_VEL
LIN {X 0,Y 520.559,Z 518.2,A -85,B 0,C 180,E1 24679.407,E2 24679.407} C_VEL
LIN {X 0,Y 520.585,Z 518.192,A -85,B 0,C 180,E1 24675.941,E2 24675.941} C_VEL
LIN {X 0,Y 520.58,Z 518.188,A -85,B 0,C 180,E1 24672.422,E2 24672.422} C_VEL
LIN {X 0,Y 520.568,Z 518.191,A -85,B 0,C 180,E1 24668.95,E2 24668.95} C_VEL
LIN {X 0,Y 520.577,Z 518.193,A -85,B 0,C 180,E1 24665.511,E2 24665.511} C_VEL
LIN {X 0,Y 520.577,Z 518.198,A -85,B 0,C 180,E1 24661.981,E2 24661.981} C_VEL
LIN {X 0,Y 520.578,Z 518.198,A -85,B 0,C 180,E1 24658.569,E2 24658.569} C_VEL
LIN {X 0,Y 520.563,Z 518.195,A -85,B 0,C 180,E1 24655.152,E2 24655.152} C_VEL
LIN {X 0,Y 520.58,Z 518.196,A -85,B 0,C 180,E1 24651.718,E2 24651.718} C_VEL
LIN {X 0,Y 520.583,Z 518.18,A -85,B 0,C 180,E1 24648.253,E2 24648.253} C_VEL
LIN {X 0,Y 520.55,Z 518.198,A -85,B 0,C 180,E1 24644.857,E2 24644.857} C_VEL
LIN {X 0,Y 520.581,Z 518.182,A -85,B 0,C 180,E1 24641.408,E2 24641.408} C_VEL
LIN {X 0,Y 520.564,Z 518.198,A -85,B 0,C 180,E1 24638.004,E2 24638.004} C_VEL
LIN {X 0,Y 520.54,Z 518.203,A -85,B 0,C 180,E1 24634.516,E2 24634.516} C_VEL
LIN {X 0,Y 520.589,Z 518.184,A -85,B 0,C 180,E1 24631.142,E2 24631.142} C_VEL
LIN {X 0,Y 520.532,Z 518.205,A -85,B 0,C 180,E1 24627.854,E2 24627.854} C_VEL
LIN {X 0,Y 520.548,Z 518.192,A -85,B 0,C 180,E1 24624.409,E2 24624.409} C_VEL
LIN {X 0,Y 520.539,Z 518.192,A -85,B 0,C 180,E1 24621.231,E2 24621.231} C_VEL
LIN {X 0,Y 520.523,Z 518.206,A -85,B 0,C 180,E1 24617.872,E2 24617.872} C_VEL
LIN {X 0,Y 519.733,Z 518.304,A -85,B 0,C 180,E1 24617.549,E2 24617.549} C_VEL
LIN {X 0,Y 513.211,Z 519.123,A -85,B 0,C 180,E1 24616.563,E2 24616.563} C_VEL
LIN {X 0,Y 512.627,Z 519.195,A -85,B 0,C 180,E1 24616.285,E2 24616.285} C_VEL
LIN {X 0,Y 512.606,Z 519.315,A -85,B 0,C 180,E1 24615.896,E2 24615.896} C_VEL
LIN {X 0,Y 513.761,Z 522.495,A -85,B 0,C 180,E1 24615.699,E2 24615.699} C_VEL
LIN {X 0,Y 516.373,Z 525.493,A -85,B 0,C 180,E1 24615.341,E2 24615.341} C_VEL
LIN {X 0,Y 519.016,Z 529.36,A -85,B 0,C 180,E1 24614.969,E2 24614.969} C_VEL
LIN {X 0,Y 530.207,Z 545.408,A -85,B 0,C 180,E1 24613.465,E2 24613.465} C_VEL
LIN {X 0,Y 533.818,Z 551.151,A -85,B 0,C 180,E1 24612.991,E2 24612.991} C_VEL
LIN {X 0,Y 530.967,Z 737.878,A -85,B 0,C 180,E1 24609.96,E2 24609.96} C_VEL
LIN {X 0,Y 529.047,Z 862.503,A -85,B 0,C 180,E1 24607.961,E2 24607.961} C_VEL
LIN {X 0,Y 528.187,Z 885.438,A -85,B 0,C 180,E1 24607.407,E2 24607.407} C_VEL
LIN {X 0,Y 527.191,Z 906.062,A -85,B 0,C 180,E1 24606.737,E2 24606.737} C_VEL
LIN {X 0,Y 525.912,Z 927.515,A -85,B 0,C 180,E1 24605.844,E2 24605.844} C_VEL
LIN {X 0,Y 524.579,Z 947.927,A -85,B 0,C 180,E1 24604.804,E2 24604.804} C_VEL
LIN {X 0,Y 522.943,Z 969.513,A -85,B 0,C 180,E1 24603.478,E2 24603.478} C_VEL
LIN {X 0,Y 521.407,Z 989.292,A -85,B 0,C 180,E1 24602.05,E2 24602.05} C_VEL
LIN {X 0,Y 519.763,Z 1008.789,A -85,B 0,C 180,E1 24600.393,E2 24600.393} C_VEL
LIN {X 0,Y 518.192,Z 1027.831,A -85,B 0,C 180,E1 24598.526,E2 24598.526} C_VEL
LIN {X 0,Y 516.817,Z 1044.483,A -85,B 0,C 180,E1 24596.644,E2 24596.644} C_VEL
LIN {X 0,Y 515.557,Z 1060.831,A -85,B 0,C 180,E1 24594.521,E2 24594.521} C_VEL
LIN {X 0,Y 514.488,Z 1075.953,A -85,B 0,C 180,E1 24592.27,E2 24592.27} C_VEL
LIN {X 0,Y 513.649,Z 1088.849,A -85,B 0,C 180,E1 24590.036,E2 24590.036} C_VEL
LIN {X 0,Y 512.956,Z 1101.607,A -85,B 0,C 180,E1 24587.469,E2 24587.469} C_VEL
LIN {X 0,Y 512.521,Z 1111.351,A -85,B 0,C 180,E1 24585.154,E2 24585.154} C_VEL
LIN {X 0,Y 512.187,Z 1120.42,A -85,B 0,C 180,E1 24582.56,E2 24582.56} C_VEL
LIN {X 0,Y 512.033,Z 1127.125,A -85,B 0,C 180,E1 24580.207,E2 24580.207} C_VEL
LIN {X 0,Y 511.946,Z 1132.759,A -85,B 0,C 180,E1 24577.632,E2 24577.632} C_VEL
LIN {X 0,Y 511.907,Z 1136.372,A -85,B 0,C 180,E1 24575.38,E2 24575.38} C_VEL
LIN {X 0,Y 511.894,Z 1138.959,A -85,B 0,C 180,E1 24572.799,E2 24572.799} C_VEL
LIN {X 0,Y 511.887,Z 1139.886,A -85,B 0,C 180,E1 24570.56,E2 24570.56} C_VEL
LIN {X 0,Y 511.91,Z 1139.486,A -85,B 0,C 180,E1 24567.985,E2 24567.985} C_VEL
LIN {X 0,Y 511.91,Z 1137.662,A -85,B 0,C 180,E1 24565.632,E2 24565.632} C_VEL
LIN {X 0,Y 511.915,Z 1134.164,A -85,B 0,C 180,E1 24563.045,E2 24563.045} C_VEL
LIN {X 0,Y 511.997,Z 1129.675,A -85,B 0,C 180,E1 24560.785,E2 24560.785} C_VEL
LIN {X 0,Y 512.131,Z 1123.315,A -85,B 0,C 180,E1 24558.285,E2 24558.285} C_VEL
LIN {X 0,Y 512.35,Z 1115.502,A -85,B 0,C 180,E1 24555.881,E2 24555.881} C_VEL
LIN {X 0,Y 512.74,Z 1106.135,A -85,B 0,C 180,E1 24553.459,E2 24553.459} C_VEL
LIN {X 0,Y 513.263,Z 1095.373,A -85,B 0,C 180,E1 24551.133,E2 24551.133} C_VEL
LIN {X 0,Y 514.058,Z 1082.122,A -85,B 0,C 180,E1 24548.671,E2 24548.671} C_VEL
LIN {X 0,Y 514.97,Z 1068.856,A -85,B 0,C 180,E1 24546.545,E2 24546.545} C_VEL
LIN {X 0,Y 516.185,Z 1052.602,A -85,B 0,C 180,E1 24544.285,E2 24544.285} C_VEL
LIN {X 0,Y 517.536,Z 1035.835,A -85,B 0,C 180,E1 24542.251,E2 24542.251} C_VEL
LIN {X 0,Y 519.006,Z 1018.004,A -85,B 0,C 180,E1 24540.387,E2 24540.387} C_VEL
LIN {X 0,Y 520.65,Z 998.045,A -85,B 0,C 180,E1 24538.575,E2 24538.575} C_VEL
LIN {X 0,Y 522.264,Z 978.65,A -85,B 0,C 180,E1 24537.064,E2 24537.064} C_VEL
LIN {X 0,Y 523.841,Z 957.503,A -85,B 0,C 180,E1 24535.666,E2 24535.666} C_VEL
LIN {X 0,Y 525.355,Z 936.908,A -85,B 0,C 180,E1 24534.516,E2 24534.516} C_VEL
LIN {X 0,Y 526.61,Z 916.398,A -85,B 0,C 180,E1 24533.582,E2 24533.582} C_VEL
LIN {X 0,Y 527.738,Z 895.577,A -85,B 0,C 180,E1 24532.807,E2 24532.807} C_VEL
LIN {X 0,Y 528.664,Z 872.706,A -85,B 0,C 180,E1 24532.171,E2 24532.171} C_VEL
LIN {X 0,Y 529.362,Z 849.001,A -85,B 0,C 180,E1 24531.71,E2 24531.71} C_VEL
LIN {X 0,Y 532.353,Z 644.853,A -85,B 0,C 180,E1 24528.453,E2 24528.453} C_VEL
LIN {X 0,Y 533.711,Z 550.689,A -85,B 0,C 180,E1 24526.9,E2 24526.9} C_VEL
LIN {X 0,Y 524.975,Z 537.922,A -85,B 0,C 180,E1 24525.755,E2 24525.755} C_VEL
LIN {X 0,Y 518.903,Z 529.262,A -85,B 0,C 180,E1 24524.927,E2 24524.927} C_VEL
LIN {X 0,Y 516.27,Z 525.292,A -85,B 0,C 180,E1 24524.553,E2 24524.553} C_VEL
LIN {X 0,Y 513.358,Z 521.783,A -85,B 0,C 180,E1 24524.15,E2 24524.15} C_VEL
LIN {X 0,Y 512.59,Z 519.2,A -85,B 0,C 180,E1 24523.981,E2 24523.981} C_VEL
LIN {X 0,Y 512.574,Z 519.196,A -85,B 0,C 180,E1 24520.509,E2 24520.509} C_VEL
LIN {X 0,Y 512.642,Z 519.191,A -85,B 0,C 180,E1 24517.202,E2 24517.202} C_VEL
LIN {X 0,Y 512.585,Z 519.178,A -85,B 0,C 180,E1 24513.802,E2 24513.802} C_VEL
LIN {X 0,Y 512.607,Z 519.179,A -85,B 0,C 180,E1 24510.344,E2 24510.344} C_VEL
LIN {X 0,Y 512.629,Z 519.19,A -85,B 0,C 180,E1 24507.03,E2 24507.03} C_VEL
LIN {X 0,Y 512.594,Z 519.168,A -85,B 0,C 180,E1 24503.57,E2 24503.57} C_VEL
LIN {X 0,Y 512.646,Z 519.189,A -85,B 0,C 180,E1 24500.195,E2 24500.195} C_VEL
LIN {X 0,Y 512.621,Z 519.165,A -85,B 0,C 180,E1 24496.727,E2 24496.727} C_VEL
LIN {X 0,Y 512.615,Z 519.19,A -85,B 0,C 180,E1 24493.269,E2 24493.269} C_VEL
LIN {X 0,Y 512.644,Z 519.189,A -85,B 0,C 180,E1 24489.883,E2 24489.883} C_VEL
LIN {X 0,Y 512.622,Z 519.193,A -85,B 0,C 180,E1 24486.496,E2 24486.496} C_VEL
LIN {X 0,Y 512.63,Z 519.189,A -85,B 0,C 180,E1 24482.907,E2 24482.907} C_VEL
LIN {X 0,Y 512.638,Z 519.191,A -85,B 0,C 180,E1 24479.441,E2 24479.441} C_VEL
LIN {X 0,Y 512.634,Z 519.19,A -85,B 0,C 180,E1 24475.974,E2 24475.974} C_VEL
LIN {X 0,Y 512.64,Z 519.187,A -85,B 0,C 180,E1 24472.379,E2 24472.379} C_VEL
LIN {X 0,Y 512.627,Z 519.163,A -85,B 0,C 180,E1 24468.867,E2 24468.867} C_VEL
LIN {X 0,Y 512.649,Z 519.194,A -85,B 0,C 180,E1 24465.313,E2 24465.313} C_VEL
LIN {X 0,Y 512.642,Z 519.163,A -85,B 0,C 180,E1 24461.777,E2 24461.777} C_VEL
LIN {X 0,Y 512.621,Z 519.188,A -85,B 0,C 180,E1 24458.368,E2 24458.368} C_VEL
LIN {X 0,Y 512.639,Z 519.18,A -85,B 0,C 180,E1 24454.822,E2 24454.822} C_VEL
LIN {X 0,Y 512.65,Z 519.171,A -85,B 0,C 180,E1 24451.329,E2 24451.329} C_VEL
LIN {X 0,Y 512.607,Z 519.192,A -85,B 0,C 180,E1 24447.958,E2 24447.958} C_VEL
LIN {X 0,Y 512.644,Z 519.182,A -85,B 0,C 180,E1 24444.601,E2 24444.601} C_VEL
LIN {X 0,Y 512.608,Z 519.175,A -85,B 0,C 180,E1 24441.236,E2 24441.236} C_VEL
LIN {X 0,Y 512.648,Z 519.403,A -85,B 0,C 180,E1 24437.996,E2 24437.996} C_VEL
LIN {X 0,Y 513.944,Z 522.728,A -85,B 0,C 180,E1 24437.541,E2 24437.541} C_VEL
LIN {X 0,Y 515.108,Z 525.015,A -85,B 0,C 180,E1 24437.199,E2 24437.199} C_VEL
LIN {X 0,Y 519.294,Z 533.638,A -85,B 0,C 180,E1 24435.967,E2 24435.967} C_VEL
LIN {X 0,Y 523.66,Z 542.562,A -85,B 0,C 180,E1 24434.781,E2 24434.781} C_VEL
LIN {X 0,Y 532.392,Z 556.229,A -85,B 0,C 180,E1 24433.616,E2 24433.616} C_VEL
LIN {X 0,Y 534.042,Z 565.176,A -85,B 0,C 180,E1 24433.287,E2 24433.287} C_VEL
LIN {X 0,Y 531.235,Z 748.95,A -85,B 0,C 180,E1 24430.309,E2 24430.309} C_VEL
LIN {X 0,Y 529.052,Z 892.294,A -85,B 0,C 180,E1 24428.009,E2 24428.009} C_VEL
LIN {X 0,Y 528.198,Z 915.223,A -85,B 0,C 180,E1 24427.458,E2 24427.458} C_VEL
LIN {X 0,Y 527.215,Z 935.601,A -85,B 0,C 180,E1 24426.798,E2 24426.798} C_VEL
LIN {X 0,Y 525.859,Z 958.387,A -85,B 0,C 180,E1 24425.847,E2 24425.847} C_VEL
LIN {X 0,Y 524.537,Z 978.578,A -85,B 0,C 180,E1 24424.813,E2 24424.813} C_VEL
LIN {X 0,Y 522.891,Z 1000.137,A -85,B 0,C 180,E1 24423.481,E2 24423.481} C_VEL
LIN {X 0,Y 521.357,Z 1019.974,A -85,B 0,C 180,E1 24422.042,E2 24422.042} C_VEL
LIN {X 0,Y 519.723,Z 1039.27,A -85,B 0,C 180,E1 24420.396,E2 24420.396} C_VEL
LIN {X 0,Y 518.081,Z 1059.135,A -85,B 0,C 180,E1 24418.43,E2 24418.43} C_VEL
LIN {X 0,Y 516.728,Z 1075.66,A -85,B 0,C 180,E1 24416.55,E2 24416.55} C_VEL
LIN {X 0,Y 515.53,Z 1091.146,A -85,B 0,C 180,E1 24414.522,E2 24414.522} C_VEL
LIN {X 0,Y 514.469,Z 1106.221,A -85,B 0,C 180,E1 24412.27,E2 24412.27} C_VEL
LIN {X 0,Y 513.635,Z 1119.091,A -85,B 0,C 180,E1 24410.036,E2 24410.036} C_VEL
LIN {X 0,Y 512.946,Z 1131.807,A -85,B 0,C 180,E1 24407.469,E2 24407.469} C_VEL
LIN {X 0,Y 512.516,Z 1141.53,A -85,B 0,C 180,E1 24405.154,E2 24405.154} C_VEL
LIN {X 0,Y 512.193,Z 1150.346,A -85,B 0,C 180,E1 24402.629,E2 24402.629} C_VEL
LIN {X 0,Y 512.043,Z 1156.867,A -85,B 0,C 180,E1 24400.349,E2 24400.349} C_VEL
LIN {X 0,Y 511.954,Z 1162.635,A -85,B 0,C 180,E1 24397.744,E2 24397.744} C_VEL
LIN {X 0,Y 511.906,Z 1166.278,A -85,B 0,C 180,E1 24395.492,E2 24395.492} C_VEL
LIN {X 0,Y 511.891,Z 1168.919,A -85,B 0,C 180,E1 24392.911,E2 24392.911} C_VEL
LIN {X 0,Y 511.884,Z 1169.872,A -85,B 0,C 180,E1 24390.671,E2 24390.671} C_VEL
LIN {X 0,Y 511.906,Z 1169.526,A -85,B 0,C 180,E1 24388.097,E2 24388.097} C_VEL
LIN {X 0,Y 511.915,Z 1167.729,A -85,B 0,C 180,E1 24385.743,E2 24385.743} C_VEL
LIN {X 0,Y 511.925,Z 1164.493,A -85,B 0,C 180,E1 24383.27,E2 24383.27} C_VEL
LIN {X 0,Y 511.998,Z 1159.827,A -85,B 0,C 180,E1 24380.898,E2 24380.898} C_VEL
LIN {X 0,Y 512.125,Z 1153.516,A -85,B 0,C 180,E1 24378.399,E2 24378.399} C_VEL
LIN {X 0,Y 512.354,Z 1145.423,A -85,B 0,C 180,E1 24375.904,E2 24375.904} C_VEL
LIN {X 0,Y 512.747,Z 1135.936,A -85,B 0,C 180,E1 24373.459,E2 24373.459} C_VEL
LIN {X 0,Y 513.277,Z 1125.151,A -85,B 0,C 180,E1 24371.133,E2 24371.133} C_VEL
LIN {X 0,Y 514.074,Z 1111.856,A -85,B 0,C 180,E1 24368.671,E2 24368.671} C_VEL
LIN {X 0,Y 514.993,Z 1098.563,A -85,B 0,C 180,E1 24366.546,E2 24366.546} C_VEL
LIN {X 0,Y 516.178,Z 1082.723,A -85,B 0,C 180,E1 24364.346,E2 24364.346} C_VEL
LIN {X 0,Y 517.524,Z 1065.986,A -85,B 0,C 180,E1 24362.312,E2 24362.312} C_VEL
LIN {X 0,Y 518.991,Z 1048.173,A -85,B 0,C 180,E1 24360.449,E2 24360.449} C_VEL
LIN {X 0,Y 520.634,Z 1028.255,A -85,B 0,C 180,E1 24358.637,E2 24358.637} C_VEL
LIN {X 0,Y 522.24,Z 1008.893,A -85,B 0,C 180,E1 24357.127,E2 24357.127} C_VEL
LIN {X 0,Y 523.822,Z 987.819,A -85,B 0,C 180,E1 24355.73,E2 24355.73} C_VEL
LIN {X 0,Y 525.408,Z 966.06,A -85,B 0,C 180,E1 24354.519,E2 24354.519} C_VEL
LIN {X 0,Y 526.677,Z 945.2,A -85,B 0,C 180,E1 24353.578,E2 24353.578} C_VEL
LIN {X 0,Y 527.835,Z 923.411,A -85,B 0,C 180,E1 24352.78,E2 24352.78} C_VEL
LIN {X 0,Y 528.727,Z 901.306,A -85,B 0,C 180,E1 24352.184,E2 24352.184} C_VEL
LIN {X 0,Y 529.413,Z 875.288,A -85,B 0,C 180,E1 24351.696,E2 24351.696} C_VEL
LIN {X 0,Y 532.352,Z 674.18,A -85,B 0,C 180,E1 24348.488,E2 24348.488} C_VEL
LIN {X 0,Y 533.898,Z 563.524,A -85,B 0,C 180,E1 24346.668,E2 24346.668} C_VEL
LIN {X 0,Y 532.088,Z 555.52,A -85,B 0,C 180,E1 24346.34,E2 24346.34} C_VEL
LIN {X 0,Y 523.2,Z 541.813,A -85,B 0,C 180,E1 24345.153,E2 24345.153} C_VEL
LIN {X 0,Y 516.041,Z 526.881,A -85,B 0,C 180,E1 24343.074,E2 24343.074} C_VEL
LIN {X 0,Y 513.942,Z 522.729,A -85,B 0,C 180,E1 24342.46,E2 24342.46} C_VEL
LIN {X 0,Y 512.619,Z 519.175,A -85,B 0,C 180,E1 24341.96,E2 24341.96} C_VEL
LIN {X 0,Y 512.6,Z 519.197,A -85,B 0,C 180,E1 24338.479,E2 24338.479} C_VEL
LIN {X 0,Y 512.65,Z 519.176,A -85,B 0,C 180,E1 24335.124,E2 24335.124} C_VEL
LIN {X 0,Y 512.623,Z 519.194,A -85,B 0,C 180,E1 24331.646,E2 24331.646} C_VEL
LIN {X 0,Y 512.614,Z 519.179,A -85,B 0,C 180,E1 24328.159,E2 24328.159} C_VEL
LIN {X 0,Y 512.644,Z 519.169,A -85,B 0,C 180,E1 24324.792,E2 24324.792} C_VEL
LIN {X 0,Y 512.625,Z 519.187,A -85,B 0,C 180,E1 24321.271,E2 24321.271} C_VEL
LIN {X 0,Y 512.627,Z 519.162,A -85,B 0,C 180,E1 24317.714,E2 24317.714} C_VEL
LIN {X 0,Y 512.641,Z 519.191,A -85,B 0,C 180,E1 24314.341,E2 24314.341} C_VEL
LIN {X 0,Y 512.628,Z 519.164,A -85,B 0,C 180,E1 24310.905,E2 24310.905} C_VEL
LIN {X 0,Y 512.648,Z 519.186,A -85,B 0,C 180,E1 24307.396,E2 24307.396} C_VEL
LIN {X 0,Y 512.633,Z 519.192,A -85,B 0,C 180,E1 24303.914,E2 24303.914} C_VEL
LIN {X 0,Y 512.638,Z 519.19,A -85,B 0,C 180,E1 24300.447,E2 24300.447} C_VEL
LIN {X 0,Y 512.637,Z 519.187,A -85,B 0,C 180,E1 24296.981,E2 24296.981} C_VEL
LIN {X 0,Y 512.626,Z 519.194,A -85,B 0,C 180,E1 24293.504,E2 24293.504} C_VEL
LIN {X 0,Y 512.641,Z 519.166,A -85,B 0,C 180,E1 24290.053,E2 24290.053} C_VEL
LIN {X 0,Y 512.623,Z 519.188,A -85,B 0,C 180,E1 24286.579,E2 24286.579} C_VEL
LIN {X 0,Y 512.617,Z 519.164,A -85,B 0,C 180,E1 24283.104,E2 24283.104} C_VEL
LIN {X 0,Y 512.648,Z 519.188,A -85,B 0,C 180,E1 24279.686,E2 24279.686} C_VEL
LIN {X 0,Y 512.6,Z 519.164,A -85,B 0,C 180,E1 24276.308,E2 24276.308} C_VEL
LIN {X 0,Y 512.622,Z 519.192,A -85,B 0,C 180,E1 24272.802,E2 24272.802} C_VEL
LIN {X 0,Y 512.631,Z 519.174,A -85,B 0,C 180,E1 24269.398,E2 24269.398} C_VEL
LIN {X 0,Y 512.588,Z 519.18,A -85,B 0,C 180,E1 24265.998,E2 24265.998} C_VEL
LIN {X 0,Y 512.632,Z 519.191,A -85,B 0,C 180,E1 24262.546,E2 24262.546} C_VEL
LIN {X 0,Y 512.586,Z 519.194,A -85,B 0,C 180,E1 24259.345,E2 24259.345} C_VEL
LIN {X 0,Y 512.627,Z 519.195,A -85,B 0,C 180,E1 24256.285,E2 24256.285} C_VEL
LIN {X 0,Y 512.841,Z 520.074,A -85,B 0,C 180,E1 24256.008,E2 24256.008} C_VEL
LIN {X 0,Y 513.645,Z 523.257,A -85,B 0,C 180,E1 24255.709,E2 24255.709} C_VEL
LIN {X 0,Y 514.985,Z 530.618,A -85,B 0,C 180,E1 24255.405,E2 24255.405} C_VEL
LIN {X 0,Y 516.256,Z 536.831,A -85,B 0,C 180,E1 24255.136,E2 24255.136} C_VEL
LIN {X 0,Y 517.539,Z 539.342,A -85,B 0,C 180,E1 24254.941,E2 24254.941} C_VEL
LIN {X 0,Y 526.473,Z 552.284,A -85,B 0,C 180,E1 24253.728,E2 24253.728} C_VEL
LIN {X 0,Y 527.936,Z 554.73,A -85,B 0,C 180,E1 24253.529,E2 24253.529} C_VEL
LIN {X 0,Y 524.774,Z 742.254,A -85,B 0,C 180,E1 24250.453,E2 24250.453} C_VEL
LIN {X 0,Y 522.738,Z 862.654,A -85,B 0,C 180,E1 24248.5,E2 24248.5} C_VEL
LIN {X 0,Y 521.819,Z 885.32,A -85,B 0,C 180,E1 24247.948,E2 24247.948} C_VEL
LIN {X 0,Y 520.786,Z 905.216,A -85,B 0,C 180,E1 24247.299,E2 24247.299} C_VEL
LIN {X 0,Y 519.335,Z 927.529,A -85,B 0,C 180,E1 24246.369,E2 24246.369} C_VEL
LIN {X 0,Y 517.892,Z 947.831,A -85,B 0,C 180,E1 24245.326,E2 24245.326} C_VEL
LIN {X 0,Y 516.126,Z 969.39,A -85,B 0,C 180,E1 24243.99,E2 24243.99} C_VEL
LIN {X 0,Y 514.386,Z 989.656,A -85,B 0,C 180,E1 24242.511,E2 24242.511} C_VEL
LIN {X 0,Y 512.632,Z 1008.795,A -85,B 0,C 180,E1 24240.862,E2 24240.862} C_VEL
LIN {X 0,Y 510.891,Z 1027.8,A -85,B 0,C 180,E1 24238.976,E2 24238.976} C_VEL
LIN {X 0,Y 509.408,Z 1044.281,A -85,B 0,C 180,E1 24237.089,E2 24237.089} C_VEL
LIN {X 0,Y 507.985,Z 1060.834,A -85,B 0,C 180,E1 24234.912,E2 24234.912} C_VEL
LIN {X 0,Y 506.795,Z 1075.959,A -85,B 0,C 180,E1 24232.627,E2 24232.627} C_VEL
LIN {X 0,Y 505.824,Z 1089.486,A -85,B 0,C 180,E1 24230.238,E2 24230.238} C_VEL
LIN {X 0,Y 505.061,Z 1102.133,A -85,B 0,C 180,E1 24227.632,E2 24227.632} C_VEL
LIN {X 0,Y 504.563,Z 1112.27,A -85,B 0,C 180,E1 24225.164,E2 24225.164} C_VEL
LIN {X 0,Y 504.21,Z 1120.918,A -85,B 0,C 180,E1 24222.6,E2 24222.6} C_VEL
LIN {X 0,Y 504.024,Z 1127.942,A -85,B 0,C 180,E1 24220.054,E2 24220.054} C_VEL
LIN {X 0,Y 503.949,Z 1132.967,A -85,B 0,C 180,E1 24217.639,E2 24217.639} C_VEL
LIN {X 0,Y 503.916,Z 1136.851,A -85,B 0,C 180,E1 24215.123,E2 24215.123} C_VEL
LIN {X 0,Y 503.909,Z 1139.164,A -85,B 0,C 180,E1 24212.502,E2 24212.502} C_VEL
LIN {X 0,Y 503.911,Z 1139.997,A -85,B 0,C 180,E1 24210,E2 24210} C_VEL
LIN {X 0,Y 503.912,Z 1139.217,A -85,B 0,C 180,E1 24207.498,E2 24207.498} C_VEL
LIN {X 0,Y 503.916,Z 1136.972,A -85,B 0,C 180,E1 24204.878,E2 24204.878} C_VEL
LIN {X 0,Y 503.942,Z 1133.13,A -85,B 0,C 180,E1 24202.361,E2 24202.361} C_VEL
LIN {X 0,Y 504.018,Z 1128.143,A -85,B 0,C 180,E1 24199.946,E2 24199.946} C_VEL
LIN {X 0,Y 504.207,Z 1121.194,A -85,B 0,C 180,E1 24197.401,E2 24197.401} C_VEL
LIN {X 0,Y 504.532,Z 1113.046,A -85,B 0,C 180,E1 24194.953,E2 24194.953} C_VEL
LIN {X 0,Y 505.007,Z 1103.041,A -85,B 0,C 180,E1 24192.486,E2 24192.486} C_VEL
LIN {X 0,Y 505.718,Z 1091.231,A -85,B 0,C 180,E1 24189.999,E2 24189.999} C_VEL
LIN {X 0,Y 506.592,Z 1078.61,A -85,B 0,C 180,E1 24187.732,E2 24187.732} C_VEL
LIN {X 0,Y 507.792,Z 1063.141,A -85,B 0,C 180,E1 24185.327,E2 24185.327} C_VEL
LIN {X 0,Y 509.173,Z 1047.02,A -85,B 0,C 180,E1 24183.151,E2 24183.151} C_VEL
LIN {X 0,Y 510.715,Z 1029.732,A -85,B 0,C 180,E1 24181.146,E2 24181.146} C_VEL
LIN {X 0,Y 512.485,Z 1010.396,A -85,B 0,C 180,E1 24179.194,E2 24179.194} C_VEL
LIN {X 0,Y 514.162,Z 992.079,A -85,B 0,C 180,E1 24177.599,E2 24177.599} C_VEL
LIN {X 0,Y 515.927,Z 971.64,A -85,B 0,C 180,E1 24176.073,E2 24176.073} C_VEL
LIN {X 0,Y 517.619,Z 951.543,A -85,B 0,C 180,E1 24174.794,E2 24174.794} C_VEL
LIN {X 0,Y 519.142,Z 930.512,A -85,B 0,C 180,E1 24173.684,E2 24173.684} C_VEL
LIN {X 0,Y 520.591,Z 908.664,A -85,B 0,C 180,E1 24172.733,E2 24172.733} C_VEL
LIN {X 0,Y 521.738,Z 886.96,A -85,B 0,C 180,E1 24172.01,E2 24172.01} C_VEL
LIN {X 0,Y 522.697,Z 864.847,A -85,B 0,C 180,E1 24171.452,E2 24171.452} C_VEL
LIN {X 0,Y 523.709,Z 808.722,A -85,B 0,C 180,E1 24170.524,E2 24170.524} C_VEL
LIN {X 0,Y 527.232,Z 596.686,A -85,B 0,C 180,E1 24167.079,E2 24167.079} C_VEL
LIN {X 0,Y 527.805,Z 554.169,A -85,B 0,C 180,E1 24166.357,E2 24166.357} C_VEL
LIN {X 0,Y 514.854,Z 535.482,A -85,B 0,C 180,E1 24164.591,E2 24164.591} C_VEL
LIN {X 0,Y 511.124,Z 530.413,A -85,B 0,C 180,E1 24164.061,E2 24164.061} C_VEL
LIN {X 0,Y 508.457,Z 526.433,A -85,B 0,C 180,E1 24163.668,E2 24163.668} C_VEL
LIN {X 0,Y 505.375,Z 522.596,A -85,B 0,C 180,E1 24163.219,E2 24163.219} C_VEL
LIN {X 0,Y 504.663,Z 520.187,A -85,B 0,C 180,E1 24163.071,E2 24163.071} C_VEL
LIN {X 0,Y 504.646,Z 520.169,A -85,B 0,C 180,E1 24159.936,E2 24159.936} C_VEL
LIN {X 0,Y 504.648,Z 520.184,A -85,B 0,C 180,E1 24156.447,E2 24156.447} C_VEL
LIN {X 0,Y 504.709,Z 520.169,A -85,B 0,C 180,E1 24153.011,E2 24153.011} C_VEL
LIN {X 0,Y 504.649,Z 520.162,A -85,B 0,C 180,E1 24149.691,E2 24149.691} C_VEL
LIN {X 0,Y 504.682,Z 520.18,A -85,B 0,C 180,E1 24146.219,E2 24146.219} C_VEL
LIN {X 0,Y 504.69,Z 520.154,A -85,B 0,C 180,E1 24142.849,E2 24142.849} C_VEL
LIN {X 0,Y 504.665,Z 520.18,A -85,B 0,C 180,E1 24139.427,E2 24139.427} C_VEL
LIN {X 0,Y 504.708,Z 520.158,A -85,B 0,C 180,E1 24135.984,E2 24135.984} C_VEL
LIN {X 0,Y 504.696,Z 520.178,A -85,B 0,C 180,E1 24132.471,E2 24132.471} C_VEL
LIN {X 0,Y 504.678,Z 520.178,A -85,B 0,C 180,E1 24129.005,E2 24129.005} C_VEL
LIN {X 0,Y 504.704,Z 520.173,A -85,B 0,C 180,E1 24125.571,E2 24125.571} C_VEL
LIN {X 0,Y 504.702,Z 520.179,A -85,B 0,C 180,E1 24122.044,E2 24122.044} C_VEL
LIN {X 0,Y 504.69,Z 520.178,A -85,B 0,C 180,E1 24118.524,E2 24118.524} C_VEL
LIN {X 0,Y 504.699,Z 520.174,A -85,B 0,C 180,E1 24115,E2 24115} C_VEL
LIN {X 0,Y 504.704,Z 520.177,A -85,B 0,C 180,E1 24111.456,E2 24111.456} C_VEL
LIN {X 0,Y 504.694,Z 520.154,A -85,B 0,C 180,E1 24107.878,E2 24107.878} C_VEL
LIN {X 0,Y 504.695,Z 520.174,A -85,B 0,C 180,E1 24104.37,E2 24104.37} C_VEL
LIN {X 0,Y 504.69,Z 520.168,A -85,B 0,C 180,E1 24100.8,E2 24100.8} C_VEL
LIN {X 0,Y 504.704,Z 520.165,A -85,B 0,C 180,E1 24097.396,E2 24097.396} C_VEL
LIN {X 0,Y 504.684,Z 520.18,A -85,B 0,C 180,E1 24093.908,E2 24093.908} C_VEL
LIN {X 0,Y 504.677,Z 520.162,A -85,B 0,C 180,E1 24090.311,E2 24090.311} C_VEL
LIN {X 0,Y 504.709,Z 520.162,A -85,B 0,C 180,E1 24086.855,E2 24086.855} C_VEL
LIN {X 0,Y 504.674,Z 520.182,A -85,B 0,C 180,E1 24083.392,E2 24083.392} C_VEL
LIN {X 0,Y 504.664,Z 520.187,A -85,B 0,C 180,E1 24079.769,E2 24079.769} C_VEL
LIN {X 0,Y 504.713,Z 520.357,A -85,B 0,C 180,E1 24078.875,E2 24078.875} C_VEL
LIN {X 0,Y 506.028,Z 523.665,A -85,B 0,C 180,E1 24078.402,E2 24078.402} C_VEL
LIN {X 0,Y 507.151,Z 525.866,A -85,B 0,C 180,E1 24078.061,E2 24078.061} C_VEL
LIN {X 0,Y 513.193,Z 538.226,A -85,B 0,C 180,E1 24076.24,E2 24076.24} C_VEL
LIN {X 0,Y 515.208,Z 542.179,A -85,B 0,C 180,E1 24075.721,E2 24075.721} C_VEL
LIN {X 0,Y 527.046,Z 560.541,A -85,B 0,C 180,E1 24074.087,E2 24074.087} C_VEL
LIN {X 0,Y 528.163,Z 567.074,A -85,B 0,C 180,E1 24073.851,E2 24073.851} C_VEL
LIN {X 0,Y 525.097,Z 751.167,A -85,B 0,C 180,E1 24070.838,E2 24070.838} C_VEL
LIN {X 0,Y 522.747,Z 892.294,A -85,B 0,C 180,E1 24068.551,E2 24068.551} C_VEL
LIN {X 0,Y 521.832,Z 915.091,A -85,B 0,C 180,E1 24067.999,E2 24067.999} C_VEL
LIN {X 0,Y 520.804,Z 934.843,A -85,B 0,C 180,E1 24067.357,E2 24067.357} C_VEL
LIN {X 0,Y 519.335,Z 957.548,A -85,B 0,C 180,E1 24066.413,E2 24066.413} C_VEL
LIN {X 0,Y 517.841,Z 978.581,A -85,B 0,C 180,E1 24065.33,E2 24065.33} C_VEL
LIN {X 0,Y 516.14,Z 999.234,A -85,B 0,C 180,E1 24064.045,E2 24064.045} C_VEL
LIN {X 0,Y 514.407,Z 1019.418,A -85,B 0,C 180,E1 24062.575,E2 24062.575} C_VEL
LIN {X 0,Y 512.669,Z 1038.417,A -85,B 0,C 180,E1 24060.942,E2 24060.942} C_VEL
LIN {X 0,Y 510.956,Z 1057.122,A -85,B 0,C 180,E1 24059.096,E2 24059.096} C_VEL
LIN {X 0,Y 509.468,Z 1073.632,A -85,B 0,C 180,E1 24057.211,E2 24057.211} C_VEL
LIN {X 0,Y 508.031,Z 1090.299,A -85,B 0,C 180,E1 24055.033,E2 24055.033} C_VEL
LIN {X 0,Y 506.832,Z 1105.508,A -85,B 0,C 180,E1 24052.747,E2 24052.747} C_VEL
LIN {X 0,Y 505.852,Z 1119.089,A -85,B 0,C 180,E1 24050.357,E2 24050.357} C_VEL
LIN {X 0,Y 505.083,Z 1131.808,A -85,B 0,C 180,E1 24047.749,E2 24047.749} C_VEL
LIN {X 0,Y 504.598,Z 1141.529,A -85,B 0,C 180,E1 24045.398,E2 24045.398} C_VEL
LIN {X 0,Y 504.238,Z 1150.347,A -85,B 0,C 180,E1 24042.831,E2 24042.831} C_VEL
LIN {X 0,Y 504.07,Z 1156.867,A -85,B 0,C 180,E1 24040.515,E2 24040.515} C_VEL
LIN {X 0,Y 503.966,Z 1162.635,A -85,B 0,C 180,E1 24037.868,E2 24037.868} C_VEL
LIN {X 0,Y 503.905,Z 1166.278,A -85,B 0,C 180,E1 24035.579,E2 24035.579} C_VEL
LIN {X 0,Y 503.889,Z 1168.919,A -85,B 0,C 180,E1 24032.957,E2 24032.957} C_VEL
LIN {X 0,Y 503.884,Z 1169.872,A -85,B 0,C 180,E1 24030.682,E2 24030.682} C_VEL
LIN {X 0,Y 503.907,Z 1169.526,A -85,B 0,C 180,E1 24028.067,E2 24028.067} C_VEL
LIN {X 0,Y 503.913,Z 1167.729,A -85,B 0,C 180,E1 24025.676,E2 24025.676} C_VEL
LIN {X 0,Y 503.923,Z 1164.493,A -85,B 0,C 180,E1 24023.162,E2 24023.162} C_VEL
LIN {X 0,Y 504.002,Z 1159.827,A -85,B 0,C 180,E1 24020.753,E2 24020.753} C_VEL
LIN {X 0,Y 504.156,Z 1153.516,A -85,B 0,C 180,E1 24018.213,E2 24018.213} C_VEL
LIN {X 0,Y 504.423,Z 1145.343,A -85,B 0,C 180,E1 24015.654,E2 24015.654} C_VEL
LIN {X 0,Y 504.886,Z 1135.42,A -85,B 0,C 180,E1 24013.075,E2 24013.075} C_VEL
LIN {X 0,Y 505.496,Z 1124.572,A -85,B 0,C 180,E1 24010.711,E2 24010.711} C_VEL
LIN {X 0,Y 506.399,Z 1111.154,A -85,B 0,C 180,E1 24008.21,E2 24008.21} C_VEL
LIN {X 0,Y 507.492,Z 1097.008,A -85,B 0,C 180,E1 24005.931,E2 24005.931} C_VEL
LIN {X 0,Y 508.795,Z 1081.333,A -85,B 0,C 180,E1 24003.758,E2 24003.758} C_VEL
LIN {X 0,Y 510.308,Z 1064.327,A -85,B 0,C 180,E1 24001.695,E2 24001.695} C_VEL
LIN {X 0,Y 511.832,Z 1047.547,A -85,B 0,C 180,E1 23999.927,E2 23999.927} C_VEL
LIN {X 0,Y 513.588,Z 1028.251,A -85,B 0,C 180,E1 23998.157,E2 23998.157} C_VEL
LIN {X 0,Y 515.257,Z 1009.7,A -85,B 0,C 180,E1 23996.69,E2 23996.69} C_VEL
LIN {X 0,Y 516.986,Z 988.834,A -85,B 0,C 180,E1 23995.28,E2 23995.28} C_VEL
LIN {X 0,Y 518.606,Z 968.407,A -85,B 0,C 180,E1 23994.118,E2 23994.118} C_VEL
LIN {X 0,Y 520.086,Z 946.606,A -85,B 0,C 180,E1 23993.106,E2 23993.106} C_VEL
LIN {X 0,Y 521.311,Z 925.719,A -85,B 0,C 180,E1 23992.321,E2 23992.321} C_VEL
LIN {X 0,Y 522.327,Z 902.977,A -85,B 0,C 180,E1 23991.682,E2 23991.682} C_VEL
LIN {X 0,Y 523.078,Z 879.399,A -85,B 0,C 180,E1 23991.217,E2 23991.217} C_VEL
LIN {X 0,Y 526.264,Z 678.507,A -85,B 0,C 180,E1 23987.982,E2 23987.982} C_VEL
LIN {X 0,Y 528.029,Z 565.431,A -85,B 0,C 180,E1 23986.105,E2 23986.105} C_VEL
LIN {X 0,Y 526.741,Z 559.887,A -85,B 0,C 180,E1 23985.869,E2 23985.869} C_VEL
LIN {X 0,Y 514.762,Z 541.373,A -85,B 0,C 180,E1 23984.211,E2 23984.211} C_VEL
LIN {X 0,Y 508.263,Z 528.139,A -85,B 0,C 180,E1 23982.282,E2 23982.282} C_VEL
LIN {X 0,Y 506.459,Z 524.252,A -85,B 0,C 180,E1 23981.706,E2 23981.706} C_VEL
LIN {X 0,Y 504.796,Z 520.792,A -85,B 0,C 180,E1 23981.177,E2 23981.177} C_VEL
LIN {X 0,Y 504.682,Z 520.173,A -85,B 0,C 180,E1 23981.052,E2 23981.052} C_VEL
LIN {X 0,Y 504.689,Z 520.181,A -85,B 0,C 180,E1 23977.746,E2 23977.746} C_VEL
LIN {X 0,Y 504.663,Z 520.16,A -85,B 0,C 180,E1 23974.24,E2 23974.24} C_VEL
LIN {X 0,Y 504.711,Z 520.169,A -85,B 0,C 180,E1 23970.737,E2 23970.737} C_VEL
LIN {X 0,Y 504.706,Z 520.173,A -85,B 0,C 180,E1 23967.188,E2 23967.188} C_VEL
LIN {X 0,Y 504.674,Z 520.151,A -85,B 0,C 180,E1 23963.714,E2 23963.714} C_VEL
LIN {X 0,Y 504.706,Z 520.174,A -85,B 0,C 180,E1 23960.284,E2 23960.284} C_VEL
LIN {X 0,Y 504.704,Z 520.153,A -85,B 0,C 180,E1 23956.693,E2 23956.693} C_VEL
LIN {X 0,Y 504.689,Z 520.179,A -85,B 0,C 180,E1 23953.169,E2 23953.169} C_VEL
LIN {X 0,Y 504.701,Z 520.161,A -85,B 0,C 180,E1 23949.694,E2 23949.694} C_VEL
LIN {X 0,Y 504.7,Z 520.174,A -85,B 0,C 180,E1 23946.141,E2 23946.141} C_VEL
LIN {X 0,Y 504.696,Z 520.179,A -85,B 0,C 180,E1 23942.611,E2 23942.611} C_VEL
LIN {X 0,Y 504.702,Z 520.173,A -85,B 0,C 180,E1 23939.092,E2 23939.092} C_VEL
LIN {X 0,Y 504.688,Z 520.175,A -85,B 0,C 180,E1 23935.568,E2 23935.568} C_VEL
LIN {X 0,Y 504.705,Z 520.179,A -85,B 0,C 180,E1 23932.029,E2 23932.029} C_VEL
LIN {X 0,Y 504.697,Z 520.155,A -85,B 0,C 180,E1 23928.457,E2 23928.457} C_VEL
LIN {X 0,Y 504.675,Z 520.176,A -85,B 0,C 180,E1 23924.957,E2 23924.957} C_VEL
LIN {X 0,Y 504.705,Z 520.153,A -85,B 0,C 180,E1 23921.52,E2 23921.52} C_VEL
LIN {X 0,Y 504.679,Z 520.177,A -85,B 0,C 180,E1 23918.132,E2 23918.132} C_VEL
LIN {X 0,Y 504.663,Z 520.176,A -85,B 0,C 180,E1 23914.537,E2 23914.537} C_VEL
LIN {X 0,Y 504.709,Z 520.157,A -85,B 0,C 180,E1 23911.094,E2 23911.094} C_VEL
LIN {X 0,Y 504.658,Z 520.183,A -85,B 0,C 180,E1 23907.78,E2 23907.78} C_VEL
LIN {X 0,Y 504.657,Z 520.171,A -85,B 0,C 180,E1 23904.234,E2 23904.234} C_VEL
LIN {X 0,Y 504.687,Z 520.16,A -85,B 0,C 180,E1 23900.949,E2 23900.949} C_VEL
LIN {X 0,Y 504.638,Z 520.184,A -85,B 0,C 180,E1 23897.65,E2 23897.65} C_VEL
LIN {X 0,Y 504.708,Z 520.41,A -85,B 0,C 180,E1 23896.817,E2 23896.817} C_VEL
LIN {X 0,Y 505.995,Z 523.655,A -85,B 0,C 180,E1 23896.594,E2 23896.594} C_VEL
LIN {X 0,Y 508.485,Z 526.485,A -85,B 0,C 180,E1 23896.238,E2 23896.238} C_VEL
LIN {X 0,Y 511.076,Z 530.357,A -85,B 0,C 180,E1 23895.855,E2 23895.855} C_VEL
LIN {X 0,Y 512.933,Z 532.924,A -85,B 0,C 180,E1 23895.589,E2 23895.589} C_VEL
LIN {X 0,Y 517.539,Z 539.342,A -85,B 0,C 180,E1 23894.941,E2 23894.941} C_VEL
LIN {X 0,Y 519.744,Z 543.455,A -85,B 0,C 180,E1 23894.618,E2 23894.618} C_VEL
LIN {X 0,Y 521.328,Z 549.393,A -85,B 0,C 180,E1 23894.332,E2 23894.332} C_VEL
LIN {X 0,Y 522.089,Z 558.187,A -85,B 0,C 180,E1 23894.083,E2 23894.083} C_VEL
LIN {X 0,Y 521.82,Z 573.27,A -85,B 0,C 180,E1 23893.828,E2 23893.828} C_VEL
LIN {X 0,Y 517.906,Z 787.992,A -85,B 0,C 180,E1 23890.288,E2 23890.288} C_VEL
LIN {X 0,Y 516.454,Z 863.85,A -85,B 0,C 180,E1 23889.033,E2 23889.033} C_VEL
LIN {X 0,Y 515.451,Z 886.1,A -85,B 0,C 180,E1 23888.476,E2 23888.476} C_VEL
LIN {X 0,Y 514.3,Z 906.644,A -85,B 0,C 180,E1 23887.794,E2 23887.794} C_VEL
LIN {X 0,Y 512.713,Z 928.826,A -85,B 0,C 180,E1 23886.847,E2 23886.847} C_VEL
LIN {X 0,Y 511.063,Z 950.343,A -85,B 0,C 180,E1 23885.716,E2 23885.716} C_VEL
LIN {X 0,Y 509.241,Z 970.429,A -85,B 0,C 180,E1 23884.435,E2 23884.435} C_VEL
LIN {X 0,Y 507.358,Z 990.41,A -85,B 0,C 180,E1 23882.951,E2 23882.951} C_VEL
LIN {X 0,Y 505.482,Z 1009.338,A -85,B 0,C 180,E1 23881.294,E2 23881.294} C_VEL
LIN {X 0,Y 503.536,Z 1028.65,A -85,B 0,C 180,E1 23879.342,E2 23879.342} C_VEL
LIN {X 0,Y 501.915,Z 1045.3,A -85,B 0,C 180,E1 23877.399,E2 23877.399} C_VEL
LIN {X 0,Y 500.357,Z 1061.683,A -85,B 0,C 180,E1 23875.191,E2 23875.191} C_VEL
LIN {X 0,Y 499.057,Z 1076.674,A -85,B 0,C 180,E1 23872.873,E2 23872.873} C_VEL
LIN {X 0,Y 498.054,Z 1089.488,A -85,B 0,C 180,E1 23870.568,E2 23870.568} C_VEL
LIN {X 0,Y 497.204,Z 1102.137,A -85,B 0,C 180,E1 23867.92,E2 23867.92} C_VEL
LIN {X 0,Y 496.635,Z 1112.533,A -85,B 0,C 180,E1 23865.344,E2 23865.344} C_VEL
LIN {X 0,Y 496.252,Z 1120.954,A -85,B 0,C 180,E1 23862.793,E2 23862.793} C_VEL
LIN {X 0,Y 496.05,Z 1127.944,A -85,B 0,C 180,E1 23860.217,E2 23860.217} C_VEL
LIN {X 0,Y 495.963,Z 1132.968,A -85,B 0,C 180,E1 23857.763,E2 23857.763} C_VEL
LIN {X 0,Y 495.915,Z 1136.852,A -85,B 0,C 180,E1 23855.206,E2 23855.206} C_VEL
LIN {X 0,Y 495.907,Z 1139.164,A -85,B 0,C 180,E1 23852.543,E2 23852.543} C_VEL
LIN {X 0,Y 495.911,Z 1139.997,A -85,B 0,C 180,E1 23850,E2 23850} C_VEL
LIN {X 0,Y 495.911,Z 1139.217,A -85,B 0,C 180,E1 23847.458,E2 23847.458} C_VEL
LIN {X 0,Y 495.917,Z 1137.052,A -85,B 0,C 180,E1 23844.87,E2 23844.87} C_VEL
LIN {X 0,Y 495.954,Z 1133.128,A -85,B 0,C 180,E1 23842.237,E2 23842.237} C_VEL
LIN {X 0,Y 496.04,Z 1128.141,A -85,B 0,C 180,E1 23839.783,E2 23839.783} C_VEL
LIN {X 0,Y 496.248,Z 1121.191,A -85,B 0,C 180,E1 23837.195,E2 23837.195} C_VEL
LIN {X 0,Y 496.621,Z 1112.887,A -85,B 0,C 180,E1 23834.662,E2 23834.662} C_VEL
LIN {X 0,Y 497.178,Z 1102.521,A -85,B 0,C 180,E1 23832.08,E2 23832.08} C_VEL
LIN {X 0,Y 498.019,Z 1089.955,A -85,B 0,C 180,E1 23829.431,E2 23829.431} C_VEL
LIN {X 0,Y 499.015,Z 1077.19,A -85,B 0,C 180,E1 23827.126,E2 23827.126} C_VEL
LIN {X 0,Y 500.302,Z 1062.288,A -85,B 0,C 180,E1 23824.806,E2 23824.806} C_VEL
LIN {X 0,Y 501.847,Z 1046.013,A -85,B 0,C 180,E1 23822.598,E2 23822.598} C_VEL
LIN {X 0,Y 503.484,Z 1029.168,A -85,B 0,C 180,E1 23820.626,E2 23820.626} C_VEL
LIN {X 0,Y 505.446,Z 1009.717,A -85,B 0,C 180,E1 23818.65,E2 23818.65} C_VEL
LIN {X 0,Y 507.26,Z 991.405,A -85,B 0,C 180,E1 23817.042,E2 23817.042} C_VEL
LIN {X 0,Y 509.126,Z 971.625,A -85,B 0,C 180,E1 23815.556,E2 23815.556} C_VEL
LIN {X 0,Y 510.962,Z 951.439,A -85,B 0,C 180,E1 23814.26,E2 23814.26} C_VEL
LIN {X 0,Y 512.605,Z 930.364,A -85,B 0,C 180,E1 23813.138,E2 23813.138} C_VEL
LIN {X 0,Y 514.179,Z 908.643,A -85,B 0,C 180,E1 23812.188,E2 23812.188} C_VEL
LIN {X 0,Y 515.397,Z 887.143,A -85,B 0,C 180,E1 23811.465,E2 23811.465} C_VEL
LIN {X 0,Y 516.408,Z 865.523,A -85,B 0,C 180,E1 23810.912,E2 23810.912} C_VEL
LIN {X 0,Y 517.375,Z 818.5,A -85,B 0,C 180,E1 23810.116,E2 23810.116} C_VEL
LIN {X 0,Y 521.221,Z 606.915,A -85,B 0,C 180,E1 23806.648,E2 23806.648} C_VEL
LIN {X 0,Y 522.006,Z 558.01,A -85,B 0,C 180,E1 23805.814,E2 23805.814} C_VEL
LIN {X 0,Y 510.65,Z 541.492,A -85,B 0,C 180,E1 23804.226,E2 23804.226} C_VEL
LIN {X 0,Y 504.167,Z 532.298,A -85,B 0,C 180,E1 23803.27,E2 23803.27} C_VEL
LIN {X 0,Y 501.045,Z 528.277,A -85,B 0,C 180,E1 23802.803,E2 23802.803} C_VEL
LIN {X 0,Y 500.005,Z 526.711,A -85,B 0,C 180,E1 23802.641,E2 23802.641} C_VEL
LIN {X 0,Y 497.568,Z 523.939,A -85,B 0,C 180,E1 23802.274,E2 23802.274} C_VEL
LIN {X 0,Y 496.7,Z 521.172,A -85,B 0,C 180,E1 23802.093,E2 23802.093} C_VEL
LIN {X 0,Y 496.7,Z 521.155,A -85,B 0,C 180,E1 23798.459,E2 23798.459} C_VEL
LIN {X 0,Y 496.761,Z 521.144,A -85,B 0,C 180,E1 23795.145,E2 23795.145} C_VEL
LIN {X 0,Y 496.71,Z 521.174,A -85,B 0,C 180,E1 23791.83,E2 23791.83} C_VEL
LIN {X 0,Y 496.741,Z 521.152,A -85,B 0,C 180,E1 23788.361,E2 23788.361} C_VEL
LIN {X 0,Y 496.744,Z 521.156,A -85,B 0,C 180,E1 23785.005,E2 23785.005} C_VEL
LIN {X 0,Y 496.724,Z 521.165,A -85,B 0,C 180,E1 23781.491,E2 23781.491} C_VEL
LIN {X 0,Y 496.767,Z 521.142,A -85,B 0,C 180,E1 23778.057,E2 23778.057} C_VEL
LIN {X 0,Y 496.766,Z 521.164,A -85,B 0,C 180,E1 23774.453,E2 23774.453} C_VEL
LIN {X 0,Y 496.735,Z 521.166,A -85,B 0,C 180,E1 23770.907,E2 23770.907} C_VEL
LIN {X 0,Y 496.77,Z 521.164,A -85,B 0,C 180,E1 23767.401,E2 23767.401} C_VEL
LIN {X 0,Y 496.766,Z 521.167,A -85,B 0,C 180,E1 23763.809,E2 23763.809} C_VEL
LIN {X 0,Y 496.749,Z 521.163,A -85,B 0,C 180,E1 23760.231,E2 23760.231} C_VEL
LIN {X 0,Y 496.762,Z 521.162,A -85,B 0,C 180,E1 23756.654,E2 23756.654} C_VEL
LIN {X 0,Y 496.757,Z 521.167,A -85,B 0,C 180,E1 23753.064,E2 23753.064} C_VEL
LIN {X 0,Y 496.761,Z 521.14,A -85,B 0,C 180,E1 23749.564,E2 23749.564} C_VEL
LIN {X 0,Y 496.764,Z 521.165,A -85,B 0,C 180,E1 23745.964,E2 23745.964} C_VEL
LIN {X 0,Y 496.743,Z 521.138,A -85,B 0,C 180,E1 23742.548,E2 23742.548} C_VEL
LIN {X 0,Y 496.767,Z 521.171,A -85,B 0,C 180,E1 23739.007,E2 23739.007} C_VEL
LIN {X 0,Y 496.766,Z 521.146,A -85,B 0,C 180,E1 23735.378,E2 23735.378} C_VEL
LIN {X 0,Y 496.737,Z 521.158,A -85,B 0,C 180,E1 23731.901,E2 23731.901} C_VEL
LIN {X 0,Y 496.742,Z 521.172,A -85,B 0,C 180,E1 23728.309,E2 23728.309} C_VEL
LIN {X 0,Y 496.772,Z 521.154,A -85,B 0,C 180,E1 23724.802,E2 23724.802} C_VEL
LIN {X 0,Y 496.725,Z 521.149,A -85,B 0,C 180,E1 23721.353,E2 23721.353} C_VEL
LIN {X 0,Y 496.755,Z 521.383,A -85,B 0,C 180,E1 23719.795,E2 23719.795} C_VEL
LIN {X 0,Y 498.14,Z 524.812,A -85,B 0,C 180,E1 23719.283,E2 23719.283} C_VEL
LIN {X 0,Y 499.288,Z 526.845,A -85,B 0,C 180,E1 23718.941,E2 23718.941} C_VEL
LIN {X 0,Y 506.5,Z 541.433,A -85,B 0,C 180,E1 23716.746,E2 23716.746} C_VEL
LIN {X 0,Y 521.701,Z 564.746,A -85,B 0,C 180,E1 23714.574,E2 23714.574} C_VEL
LIN {X 0,Y 522.333,Z 569.131,A -85,B 0,C 180,E1 23714.424,E2 23714.424} C_VEL
LIN {X 0,Y 518.966,Z 754.781,A -85,B 0,C 180,E1 23711.355,E2 23711.355} C_VEL
LIN {X 0,Y 516.49,Z 892.195,A -85,B 0,C 180,E1 23709.109,E2 23709.109} C_VEL
LIN {X 0,Y 515.506,Z 915.089,A -85,B 0,C 180,E1 23708.551,E2 23708.551} C_VEL
LIN {X 0,Y 514.409,Z 934.728,A -85,B 0,C 180,E1 23707.908,E2 23707.908} C_VEL
LIN {X 0,Y 512.838,Z 957.225,A -85,B 0,C 180,E1 23706.968,E2 23706.968} C_VEL
LIN {X 0,Y 511.187,Z 978.584,A -85,B 0,C 180,E1 23705.86,E2 23705.86} C_VEL
LIN {X 0,Y 509.356,Z 999.23,A -85,B 0,C 180,E1 23704.562,E2 23704.562} C_VEL
LIN {X 0,Y 507.458,Z 1019.42,A -85,B 0,C 180,E1 23703.078,E2 23703.078} C_VEL
LIN {X 0,Y 505.556,Z 1038.597,A -85,B 0,C 180,E1 23701.408,E2 23701.408} C_VEL
LIN {X 0,Y 503.696,Z 1057.121,A -85,B 0,C 180,E1 23699.557,E2 23699.557} C_VEL
LIN {X 0,Y 502.073,Z 1073.632,A -85,B 0,C 180,E1 23697.646,E2 23697.646} C_VEL
LIN {X 0,Y 500.488,Z 1090.297,A -85,B 0,C 180,E1 23695.437,E2 23695.437} C_VEL
LIN {X 0,Y 499.165,Z 1105.508,A -85,B 0,C 180,E1 23693.116,E2 23693.116} C_VEL
LIN {X 0,Y 498.083,Z 1119.087,A -85,B 0,C 180,E1 23690.689,E2 23690.689} C_VEL
LIN {X 0,Y 497.261,Z 1131.288,A -85,B 0,C 180,E1 23688.159,E2 23688.159} C_VEL
LIN {X 0,Y 496.7,Z 1141.069,A -85,B 0,C 180,E1 23685.769,E2 23685.769} C_VEL
LIN {X 0,Y 496.287,Z 1150.348,A -85,B 0,C 180,E1 23683.041,E2 23683.041} C_VEL
LIN {X 0,Y 496.084,Z 1157.169,A -85,B 0,C 180,E1 23680.568,E2 23680.568} C_VEL
LIN {X 0,Y 495.97,Z 1162.635,A -85,B 0,C 180,E1 23677.996,E2 23677.996} C_VEL
LIN {X 0,Y 495.906,Z 1166.437,A -85,B 0,C 180,E1 23675.553,E2 23675.553} C_VEL
LIN {X 0,Y 495.892,Z 1168.987,A -85,B 0,C 180,E1 23672.889,E2 23672.889} C_VEL
LIN {X 0,Y 495.884,Z 1169.895,A -85,B 0,C 180,E1 23670.577,E2 23670.577} C_VEL
LIN {X 0,Y 495.914,Z 1169.392,A -85,B 0,C 180,E1 23667.804,E2 23667.804} C_VEL
LIN {X 0,Y 495.909,Z 1167.501,A -85,B 0,C 180,E1 23665.374,E2 23665.374} C_VEL
LIN {X 0,Y 495.924,Z 1163.874,A -85,B 0,C 180,E1 23662.702,E2 23662.702} C_VEL
LIN {X 0,Y 496.006,Z 1159.573,A -85,B 0,C 180,E1 23660.485,E2 23660.485} C_VEL
LIN {X 0,Y 496.191,Z 1153.173,A -85,B 0,C 180,E1 23657.903,E2 23657.903} C_VEL
LIN {X 0,Y 496.492,Z 1145.342,A -85,B 0,C 180,E1 23655.42,E2 23655.42} C_VEL
LIN {X 0,Y 497.004,Z 1135.419,A -85,B 0,C 180,E1 23652.798,E2 23652.798} C_VEL
LIN {X 0,Y 497.691,Z 1124.573,A -85,B 0,C 180,E1 23650.397,E2 23650.397} C_VEL
LIN {X 0,Y 498.69,Z 1111.152,A -85,B 0,C 180,E1 23647.856,E2 23647.856} C_VEL
LIN {X 0,Y 499.893,Z 1097.01,A -85,B 0,C 180,E1 23645.541,E2 23645.541} C_VEL
